LIN {X 0,Y 488.777,Z 238.159,A -85,B 0,C 180,E1 22662.377,E2 22662.377} C_VEL
LIN {X 0,Y 488.746,Z 238.162,A -85,B 0,C 180,E1 22658.896,E2 22658.896} C_VEL
LIN {X 0,Y 488.779,Z 238.165,A -85,B 0,C 180,E1 22655.464,E2 22655.464} C_VEL
LIN {X 0,Y 488.782,Z 238.16,A -85,B 0,C 180,E1 22652.066,E2 22652.066} C_VEL
LIN {X 0,Y 488.749,Z 238.168,A -85,B 0,C 180,E1 22648.693,E2 22648.693} C_VEL
LIN {X 0,Y 488.78,Z 238.161,A -85,B 0,C 180,E1 22645.199,E2 22645.199} C_VEL
LIN {X 0,Y 488.773,Z 238.339,A -85,B 0,C 180,E1 22642.587,E2 22642.587} C_VEL
LIN {X 0,Y 489.136,Z 239.814,A -85,B 0,C 180,E1 22642.324,E2 22642.324} C_VEL
LIN {X 0,Y 490.915,Z 242.687,A -85,B 0,C 180,E1 22641.893,E2 22641.893} C_VEL
LIN {X 0,Y 491.79,Z 244.203,A -85,B 0,C 180,E1 22641.677,E2 22641.677} C_VEL
LIN {X 0,Y 499.359,Z 257.943,A -85,B 0,C 180,E1 22639.854,E2 22639.854} C_VEL
LIN {X 0,Y 508.111,Z 274.612,A -85,B 0,C 180,E1 22637.887,E2 22637.887} C_VEL
LIN {X 0,Y 512.984,Z 283.87,A -85,B 0,C 180,E1 22636.871,E2 22636.871} C_VEL
LIN {X 0,Y 511.655,Z 317.826,A -85,B 0,C 180,E1 22635.138,E2 22635.138} C_VEL
LIN {X 0,Y 513.562,Z 334.327,A -85,B 0,C 180,E1 22634.709,E2 22634.709} C_VEL
LIN {X 0,Y 511.315,Z 543.157,A -85,B 0,C 180,E1 22631.464,E2 22631.464} C_VEL
LIN {X 0,Y 509.844,Z 662.422,A -85,B 0,C 180,E1 22629.623,E2 22629.623} C_VEL
LIN {X 0,Y 508.964,Z 686.115,A -85,B 0,C 180,E1 22629.075,E2 22629.075} C_VEL
LIN {X 0,Y 507.975,Z 706.125,A -85,B 0,C 180,E1 22628.445,E2 22628.445} C_VEL
LIN {X 0,Y 506.503,Z 726.844,A -85,B 0,C 180,E1 22627.586,E2 22627.586} C_VEL
LIN {X 0,Y 504.754,Z 747.351,A -85,B 0,C 180,E1 22626.529,E2 22626.529} C_VEL
LIN {X 0,Y 502.729,Z 769.086,A -85,B 0,C 180,E1 22625.172,E2 22625.172} C_VEL
LIN {X 0,Y 500.805,Z 788.03,A -85,B 0,C 180,E1 22623.78,E2 22623.78} C_VEL
LIN {X 0,Y 498.7,Z 807.609,A -85,B 0,C 180,E1 22622.092,E2 22622.092} C_VEL
LIN {X 0,Y 496.763,Z 825.728,A -85,B 0,C 180,E1 22620.292,E2 22620.292} C_VEL
LIN {X 0,Y 494.892,Z 842.616,A -85,B 0,C 180,E1 22618.344,E2 22618.344} C_VEL
LIN {X 0,Y 493.244,Z 858.757,A -85,B 0,C 180,E1 22616.224,E2 22616.224} C_VEL
LIN {X 0,Y 491.79,Z 873.438,A -85,B 0,C 180,E1 22613.991,E2 22613.991} C_VEL
LIN {X 0,Y 490.472,Z 888.188,A -85,B 0,C 180,E1 22611.4,E2 22611.4} C_VEL
LIN {X 0,Y 489.549,Z 900.169,A -85,B 0,C 180,E1 22608.948,E2 22608.948} C_VEL
LIN {X 0,Y 488.87,Z 910.696,A -85,B 0,C 180,E1 22606.393,E2 22606.393} C_VEL
LIN {X 0,Y 488.409,Z 919.928,A -85,B 0,C 180,E1 22603.736,E2 22603.736} C_VEL
LIN {X 0,Y 488.124,Z 926.96,A -85,B 0,C 180,E1 22601.22,E2 22601.22} C_VEL
LIN {X 0,Y 487.984,Z 932.811,A -85,B 0,C 180,E1 22598.601,E2 22598.601} C_VEL
LIN {X 0,Y 487.929,Z 936.802,A -85,B 0,C 180,E1 22596.116,E2 22596.116} C_VEL
LIN {X 0,Y 487.91,Z 939.633,A -85,B 0,C 180,E1 22593.523,E2 22593.523} C_VEL
LIN {X 0,Y 487.909,Z 940.827,A -85,B 0,C 180,E1 22590.938,E2 22590.938} C_VEL
LIN {X 0,Y 487.9,Z 940.713,A -85,B 0,C 180,E1 22588.472,E2 22588.472} C_VEL
LIN {X 0,Y 487.911,Z 939.068,A -85,B 0,C 180,E1 22585.886,E2 22585.886} C_VEL
LIN {X 0,Y 487.942,Z 936.159,A -85,B 0,C 180,E1 22583.41,E2 22583.41} C_VEL
LIN {X 0,Y 488.024,Z 931.334,A -85,B 0,C 180,E1 22580.684,E2 22580.684} C_VEL
LIN {X 0,Y 488.184,Z 925.576,A -85,B 0,C 180,E1 22578.237,E2 22578.237} C_VEL
LIN {X 0,Y 488.514,Z 917.389,A -85,B 0,C 180,E1 22575.49,E2 22575.49} C_VEL
LIN {X 0,Y 489.013,Z 908.38,A -85,B 0,C 180,E1 22572.998,E2 22572.998} C_VEL
LIN {X 0,Y 489.759,Z 897.294,A -85,B 0,C 180,E1 22570.438,E2 22570.438} C_VEL
LIN {X 0,Y 490.767,Z 884.879,A -85,B 0,C 180,E1 22567.97,E2 22567.97} C_VEL
LIN {X 0,Y 492.003,Z 871.11,A -85,B 0,C 180,E1 22565.634,E2 22565.634} C_VEL
LIN {X 0,Y 493.652,Z 854.64,A -85,B 0,C 180,E1 22563.213,E2 22563.213} C_VEL
LIN {X 0,Y 495.425,Z 838.034,A -85,B 0,C 180,E1 22561.094,E2 22561.094} C_VEL
LIN {X 0,Y 497.321,Z 820.28,A -85,B 0,C 180,E1 22559.146,E2 22559.146} C_VEL
LIN {X 0,Y 499.39,Z 801.44,A -85,B 0,C 180,E1 22557.344,E2 22557.344} C_VEL
LIN {X 0,Y 501.303,Z 783.123,A -85,B 0,C 180,E1 22555.843,E2 22555.843} C_VEL
LIN {X 0,Y 503.334,Z 762.823,A -85,B 0,C 180,E1 22554.405,E2 22554.405} C_VEL
LIN {X 0,Y 505.168,Z 742.786,A -85,B 0,C 180,E1 22553.22,E2 22553.22} C_VEL
LIN {X 0,Y 507.007,Z 720.529,A -85,B 0,C 180,E1 22552.13,E2 22552.13} C_VEL
LIN {X 0,Y 508.179,Z 702.238,A -85,B 0,C 180,E1 22551.421,E2 22551.421} C_VEL
LIN {X 0,Y 509.277,Z 679.493,A -85,B 0,C 180,E1 22550.738,E2 22550.738} C_VEL
LIN {X 0,Y 510.06,Z 656.392,A -85,B 0,C 180,E1 22550.262,E2 22550.262} C_VEL
LIN {X 0,Y 512.708,Z 451.853,A -85,B 0,C 180,E1 22547.063,E2 22547.063} C_VEL
LIN {X 0,Y 514.091,Z 331.525,A -85,B 0,C 180,E1 22545.127,E2 22545.127} C_VEL
LIN {X 0,Y 512.215,Z 314.996,A -85,B 0,C 180,E1 22544.646,E2 22544.646} C_VEL
LIN {X 0,Y 513.652,Z 284.11,A -85,B 0,C 180,E1 22543.022,E2 22543.022} C_VEL
LIN {X 0,Y 502.953,Z 264.154,A -85,B 0,C 180,E1 22540.697,E2 22540.697} C_VEL
LIN {X 0,Y 496.082,Z 251.794,A -85,B 0,C 180,E1 22539.106,E2 22539.106} C_VEL
LIN {X 0,Y 491.249,Z 243.037,A -85,B 0,C 180,E1 22537.928,E2 22537.928} C_VEL
LIN {X 0,Y 489.18,Z 239.919,A -85,B 0,C 180,E1 22537.451,E2 22537.451} C_VEL
LIN {X 0,Y 488.792,Z 238.366,A -85,B 0,C 180,E1 22537.192,E2 22537.192} C_VEL
LIN {X 0,Y 488.759,Z 238.166,A -85,B 0,C 180,E1 22533.632,E2 22533.632} C_VEL
LIN {X 0,Y 488.81,Z 238.16,A -85,B 0,C 180,E1 22530.212,E2 22530.212} C_VEL
LIN {X 0,Y 488.783,Z 238.164,A -85,B 0,C 180,E1 22526.877,E2 22526.877} C_VEL
LIN {X 0,Y 488.768,Z 238.162,A -85,B 0,C 180,E1 22523.382,E2 22523.382} C_VEL
LIN {X 0,Y 488.817,Z 238.157,A -85,B 0,C 180,E1 22519.974,E2 22519.974} C_VEL
LIN {X 0,Y 488.801,Z 238.162,A -85,B 0,C 180,E1 22516.519,E2 22516.519} C_VEL
LIN {X 0,Y 488.777,Z 238.159,A -85,B 0,C 180,E1 22513.125,E2 22513.125} C_VEL
LIN {X 0,Y 488.812,Z 238.151,A -85,B 0,C 180,E1 22509.621,E2 22509.621} C_VEL
LIN {X 0,Y 488.824,Z 238.145,A -85,B 0,C 180,E1 22506.106,E2 22506.106} C_VEL
LIN {X 0,Y 488.79,Z 238.161,A -85,B 0,C 180,E1 22502.58,E2 22502.58} C_VEL
LIN {X 0,Y 488.792,Z 238.158,A -85,B 0,C 180,E1 22498.946,E2 22498.946} C_VEL
LIN {X 0,Y 488.828,Z 238.148,A -85,B 0,C 180,E1 22495.425,E2 22495.425} C_VEL
LIN {X 0,Y 488.826,Z 238.145,A -85,B 0,C 180,E1 22491.887,E2 22491.887} C_VEL
LIN {X 0,Y 488.799,Z 238.159,A -85,B 0,C 180,E1 22488.317,E2 22488.317} C_VEL
LIN {X 0,Y 488.806,Z 238.152,A -85,B 0,C 180,E1 22484.701,E2 22484.701} C_VEL
LIN {X 0,Y 488.829,Z 238.139,A -85,B 0,C 180,E1 22481.146,E2 22481.146} C_VEL
LIN {X 0,Y 488.833,Z 238.155,A -85,B 0,C 180,E1 22477.513,E2 22477.513} C_VEL
LIN {X 0,Y 488.813,Z 238.153,A -85,B 0,C 180,E1 22473.893,E2 22473.893} C_VEL
LIN {X 0,Y 488.812,Z 238.14,A -85,B 0,C 180,E1 22470.331,E2 22470.331} C_VEL
LIN {X 0,Y 488.826,Z 238.15,A -85,B 0,C 180,E1 22466.759,E2 22466.759} C_VEL
LIN {X 0,Y 488.825,Z 238.159,A -85,B 0,C 180,E1 22463.109,E2 22463.109} C_VEL
LIN {X 0,Y 488.82,Z 238.146,A -85,B 0,C 180,E1 22459.545,E2 22459.545} C_VEL
LIN {X 0,Y 488.82,Z 238.144,A -85,B 0,C 180,E1 22455.938,E2 22455.938} C_VEL
LIN {X 0,Y 488.823,Z 238.149,A -85,B 0,C 180,E1 22452.406,E2 22452.406} C_VEL
LIN {X 0,Y 488.818,Z 238.155,A -85,B 0,C 180,E1 22448.75,E2 22448.75} C_VEL
LIN {X 0,Y 488.827,Z 238.159,A -85,B 0,C 180,E1 22445.227,E2 22445.227} C_VEL
LIN {X 0,Y 488.818,Z 238.156,A -85,B 0,C 180,E1 22442.166,E2 22442.166} C_VEL
LIN {X 0,Y 487.85,Z 238.282,A -85,B 0,C 180,E1 22441.263,E2 22441.263} C_VEL
LIN {X 0,Y 481.301,Z 239.095,A -85,B 0,C 180,E1 22438.658,E2 22438.658} C_VEL
LIN {X 0,Y 480.88,Z 239.147,A -85,B 0,C 180,E1 22438.062,E2 22438.062} C_VEL
LIN {X 0,Y 480.87,Z 239.147,A -85,B 0,C 180,E1 22434.397,E2 22434.397} C_VEL
LIN {X 0,Y 480.885,Z 239.102,A -85,B 0,C 180,E1 22430.828,E2 22430.828} C_VEL
LIN {X 0,Y 480.922,Z 239.375,A -85,B 0,C 180,E1 22427.453,E2 22427.453} C_VEL
LIN {X 0,Y 482.307,Z 242.751,A -85,B 0,C 180,E1 22426.935,E2 22426.935} C_VEL
LIN {X 0,Y 483.272,Z 244.312,A -85,B 0,C 180,E1 22426.684,E2 22426.684} C_VEL
LIN {X 0,Y 492.023,Z 261.807,A -85,B 0,C 180,E1 22424.231,E2 22424.231} C_VEL
LIN {X 0,Y 500.621,Z 280.446,A -85,B 0,C 180,E1 22421.866,E2 22421.866} C_VEL
LIN {X 0,Y 500.816,Z 281.709,A -85,B 0,C 180,E1 22421.751,E2 22421.751} C_VEL
LIN {X 0,Y 497.054,Z 336.618,A -85,B 0,C 180,E1 22418.038,E2 22418.038} C_VEL
LIN {X 0,Y 493.768,Z 391.282,A -85,B 0,C 180,E1 22414.414,E2 22414.414} C_VEL
LIN {X 0,Y 492.829,Z 410.278,A -85,B 0,C 180,E1 22413.199,E2 22413.199} C_VEL
LIN {X 0,Y 495.7,Z 434.594,A -85,B 0,C 180,E1 22412.525,E2 22412.525} C_VEL
LIN {X 0,Y 491.917,Z 630.288,A -85,B 0,C 180,E1 22409.324,E2 22409.324} C_VEL
LIN {X 0,Y 491.137,Z 649.987,A -85,B 0,C 180,E1 22408.784,E2 22408.784} C_VEL
LIN {X 0,Y 490.201,Z 668.181,A -85,B 0,C 180,E1 22408.068,E2 22408.068} C_VEL
LIN {X 0,Y 489.059,Z 686.203,A -85,B 0,C 180,E1 22407.13,E2 22407.13} C_VEL
LIN {X 0,Y 487.793,Z 703.294,A -85,B 0,C 180,E1 22406.005,E2 22406.005} C_VEL
LIN {X 0,Y 486.482,Z 719.42,A -85,B 0,C 180,E1 22404.695,E2 22404.695} C_VEL
LIN {X 0,Y 485.186,Z 734.576,A -85,B 0,C 180,E1 22403.196,E2 22403.196} C_VEL
LIN {X 0,Y 483.987,Z 748.249,A -85,B 0,C 180,E1 22401.567,E2 22401.567} C_VEL
LIN {X 0,Y 482.969,Z 760.177,A -85,B 0,C 180,E1 22399.866,E2 22399.866} C_VEL
LIN {X 0,Y 482.049,Z 771.527,A -85,B 0,C 180,E1 22397.909,E2 22397.909} C_VEL
LIN {X 0,Y 481.356,Z 780.906,A -85,B 0,C 180,E1 22395.935,E2 22395.935} C_VEL
LIN {X 0,Y 480.854,Z 788.964,A -85,B 0,C 180,E1 22393.823,E2 22393.823} C_VEL
LIN {X 0,Y 480.512,Z 795.528,A -85,B 0,C 180,E1 22391.593,E2 22391.593} C_VEL
LIN {X 0,Y 480.321,Z 800.233,A -85,B 0,C 180,E1 22389.404,E2 22389.404} C_VEL
LIN {X 0,Y 480.24,Z 803.322,A -85,B 0,C 180,E1 22387.218,E2 22387.218} C_VEL
LIN {X 0,Y 480.207,Z 804.897,A -85,B 0,C 180,E1 22384.92,E2 22384.92} C_VEL
LIN {X 0,Y 480.214,Z 804.804,A -85,B 0,C 180,E1 22382.605,E2 22382.605} C_VEL
LIN {X 0,Y 480.271,Z 803.027,A -85,B 0,C 180,E1 22380.3,E2 22380.3} C_VEL
LIN {X 0,Y 480.393,Z 799.715,A -85,B 0,C 180,E1 22378.087,E2 22378.087} C_VEL
LIN {X 0,Y 480.645,Z 794.619,A -85,B 0,C 180,E1 22375.831,E2 22375.831} C_VEL
LIN {X 0,Y 481.023,Z 788.019,A -85,B 0,C 180,E1 22373.674,E2 22373.674} C_VEL
LIN {X 0,Y 481.584,Z 780.027,A -85,B 0,C 180,E1 22371.629,E2 22371.629} C_VEL
LIN {X 0,Y 482.373,Z 770.427,A -85,B 0,C 180,E1 22369.646,E2 22369.646} C_VEL
LIN {X 0,Y 483.334,Z 759.291,A -85,B 0,C 180,E1 22367.756,E2 22367.756} C_VEL
LIN {X 0,Y 484.484,Z 746.941,A -85,B 0,C 180,E1 22366.019,E2 22366.019} C_VEL
LIN {X 0,Y 485.754,Z 733.257,A -85,B 0,C 180,E1 22364.413,E2 22364.413} C_VEL
LIN {X 0,Y 487.102,Z 718.333,A -85,B 0,C 180,E1 22362.959,E2 22362.959} C_VEL
LIN {X 0,Y 488.479,Z 702.16,A -85,B 0,C 180,E1 22361.662,E2 22361.662} C_VEL
LIN {X 0,Y 489.815,Z 685.013,A -85,B 0,C 180,E1 22360.55,E2 22360.55} C_VEL
LIN {X 0,Y 490.966,Z 667.907,A -85,B 0,C 180,E1 22359.667,E2 22359.667} C_VEL
LIN {X 0,Y 491.994,Z 648.972,A -85,B 0,C 180,E1 22358.927,E2 22358.927} C_VEL
LIN {X 0,Y 492.809,Z 629.599,A -85,B 0,C 180,E1 22358.405,E2 22358.405} C_VEL
LIN {X 0,Y 497.37,Z 433.399,A -85,B 0,C 180,E1 22355.09,E2 22355.09} C_VEL
LIN {X 0,Y 494.063,Z 406.293,A -85,B 0,C 180,E1 22354.235,E2 22354.235} C_VEL
LIN {X 0,Y 497.804,Z 348.948,A -85,B 0,C 180,E1 22350.407,E2 22350.407} C_VEL
LIN {X 0,Y 501.905,Z 294.511,A -85,B 0,C 180,E1 22346.693,E2 22346.693} C_VEL
LIN {X 0,Y 502.643,Z 283.159,A -85,B 0,C 180,E1 22345.888,E2 22345.888} C_VEL
LIN {X 0,Y 494.295,Z 265.385,A -85,B 0,C 180,E1 22343.483,E2 22343.483} C_VEL
LIN {X 0,Y 487.623,Z 252.482,A -85,B 0,C 180,E1 22341.532,E2 22341.532} C_VEL
LIN {X 0,Y 485.062,Z 247.71,A -85,B 0,C 180,E1 22340.765,E2 22340.765} C_VEL
LIN {X 0,Y 482.927,Z 243.642,A -85,B 0,C 180,E1 22340.101,E2 22340.101} C_VEL
LIN {X 0,Y 481.112,Z 240.487,A -85,B 0,C 180,E1 22339.547,E2 22339.547} C_VEL
LIN {X 0,Y 480.861,Z 239.171,A -85,B 0,C 180,E1 22339.226,E2 22339.226} C_VEL
LIN {X 0,Y 480.812,Z 239.157,A -85,B 0,C 180,E1 22335.808,E2 22335.808} C_VEL
LIN {X 0,Y 480.823,Z 239.15,A -85,B 0,C 180,E1 22332.226,E2 22332.226} C_VEL
LIN {X 0,Y 480.874,Z 239.15,A -85,B 0,C 180,E1 22328.73,E2 22328.73} C_VEL
LIN {X 0,Y 480.814,Z 239.15,A -85,B 0,C 180,E1 22325.369,E2 22325.369} C_VEL
LIN {X 0,Y 480.812,Z 239.153,A -85,B 0,C 180,E1 22321.787,E2 22321.787} C_VEL
LIN {X 0,Y 480.871,Z 239.149,A -85,B 0,C 180,E1 22318.451,E2 22318.451} C_VEL
LIN {X 0,Y 480.822,Z 239.155,A -85,B 0,C 180,E1 22314.896,E2 22314.896} C_VEL
LIN {X 0,Y 480.807,Z 239.15,A -85,B 0,C 180,E1 22311.389,E2 22311.389} C_VEL
LIN {X 0,Y 480.846,Z 239.145,A -85,B 0,C 180,E1 22307.876,E2 22307.876} C_VEL
LIN {X 0,Y 480.836,Z 239.146,A -85,B 0,C 180,E1 22304.44,E2 22304.44} C_VEL
LIN {X 0,Y 480.809,Z 239.155,A -85,B 0,C 180,E1 22300.944,E2 22300.944} C_VEL
LIN {X 0,Y 480.828,Z 239.149,A -85,B 0,C 180,E1 22297.405,E2 22297.405} C_VEL
LIN {X 0,Y 480.862,Z 239.145,A -85,B 0,C 180,E1 22293.926,E2 22293.926} C_VEL
LIN {X 0,Y 480.813,Z 239.157,A -85,B 0,C 180,E1 22290.472,E2 22290.472} C_VEL
LIN {X 0,Y 480.814,Z 239.154,A -85,B 0,C 180,E1 22286.844,E2 22286.844} C_VEL
LIN {X 0,Y 480.9,Z 239.379,A -85,B 0,C 180,E1 22283.571,E2 22283.571} C_VEL
LIN {X 0,Y 481.418,Z 241.262,A -85,B 0,C 180,E1 22283.262,E2 22283.262} C_VEL
LIN {X 0,Y 483.785,Z 245.048,A -85,B 0,C 180,E1 22282.657,E2 22282.657} C_VEL
LIN {X 0,Y 489.175,Z 254.643,A -85,B 0,C 180,E1 22281.284,E2 22281.284} C_VEL
LIN {X 0,Y 498.036,Z 270.886,A -85,B 0,C 180,E1 22279.186,E2 22279.186} C_VEL
LIN {X 0,Y 506.549,Z 287.807,A -85,B 0,C 180,E1 22277.268,E2 22277.268} C_VEL
LIN {X 0,Y 505.185,Z 318.867,A -85,B 0,C 180,E1 22275.661,E2 22275.661} C_VEL
LIN {X 0,Y 507.064,Z 335.609,A -85,B 0,C 180,E1 22275.219,E2 22275.219} C_VEL
LIN {X 0,Y 504.613,Z 544.405,A -85,B 0,C 180,E1 22271.943,E2 22271.943} C_VEL
LIN {X 0,Y 503.059,Z 661.873,A -85,B 0,C 180,E1 22270.114,E2 22270.114} C_VEL
LIN {X 0,Y 502.137,Z 685.477,A -85,B 0,C 180,E1 22269.566,E2 22269.566} C_VEL
LIN {X 0,Y 501.063,Z 706.219,A -85,B 0,C 180,E1 22268.91,E2 22268.91} C_VEL
LIN {X 0,Y 499.518,Z 729.104,A -85,B 0,C 180,E1 22267.979,E2 22267.979} C_VEL
LIN {X 0,Y 497.975,Z 749.576,A -85,B 0,C 180,E1 22266.953,E2 22266.953} C_VEL
LIN {X 0,Y 495.997,Z 769.437,A -85,B 0,C 180,E1 22265.694,E2 22265.694} C_VEL
LIN {X 0,Y 493.89,Z 788.838,A -85,B 0,C 180,E1 22264.248,E2 22264.248} C_VEL
LIN {X 0,Y 491.613,Z 808.274,A -85,B 0,C 180,E1 22262.542,E2 22262.542} C_VEL
LIN {X 0,Y 489.506,Z 826.577,A -85,B 0,C 180,E1 22260.691,E2 22260.691} C_VEL
LIN {X 0,Y 487.454,Z 843.629,A -85,B 0,C 180,E1 22258.682,E2 22258.682} C_VEL
LIN {X 0,Y 485.566,Z 860.525,A -85,B 0,C 180,E1 22256.397,E2 22256.397} C_VEL
LIN {X 0,Y 483.993,Z 875.458,A -85,B 0,C 180,E1 22254.062,E2 22254.062} C_VEL
LIN {X 0,Y 482.68,Z 888.821,A -85,B 0,C 180,E1 22251.635,E2 22251.635} C_VEL
LIN {X 0,Y 481.687,Z 900.731,A -85,B 0,C 180,E1 22249.144,E2 22249.144} C_VEL
LIN {X 0,Y 480.948,Z 911.153,A -85,B 0,C 180,E1 22246.546,E2 22246.546} C_VEL
LIN {X 0,Y 480.447,Z 920.285,A -85,B 0,C 180,E1 22243.845,E2 22243.845} C_VEL
LIN {X 0,Y 480.154,Z 926.96,A -85,B 0,C 180,E1 22241.408,E2 22241.408} C_VEL
LIN {X 0,Y 479.991,Z 932.811,A -85,B 0,C 180,E1 22238.745,E2 22238.745} C_VEL
LIN {X 0,Y 479.934,Z 936.801,A -85,B 0,C 180,E1 22236.218,E2 22236.218} C_VEL
LIN {X 0,Y 479.911,Z 939.633,A -85,B 0,C 180,E1 22233.582,E2 22233.582} C_VEL
LIN {X 0,Y 479.909,Z 940.827,A -85,B 0,C 180,E1 22230.954,E2 22230.954} C_VEL
LIN {X 0,Y 479.899,Z 940.713,A -85,B 0,C 180,E1 22228.447,E2 22228.447} C_VEL
LIN {X 0,Y 479.91,Z 939.068,A -85,B 0,C 180,E1 22225.817,E2 22225.817} C_VEL
LIN {X 0,Y 479.944,Z 936.159,A -85,B 0,C 180,E1 22223.299,E2 22223.299} C_VEL
LIN {X 0,Y 480.036,Z 931.334,A -85,B 0,C 180,E1 22220.528,E2 22220.528} C_VEL
LIN {X 0,Y 480.207,Z 925.738,A -85,B 0,C 180,E1 22218.103,E2 22218.103} C_VEL
LIN {X 0,Y 480.573,Z 917.552,A -85,B 0,C 180,E1 22215.295,E2 22215.295} C_VEL
LIN {X 0,Y 481.101,Z 908.845,A -85,B 0,C 180,E1 22212.835,E2 22212.835} C_VEL
LIN {X 0,Y 481.914,Z 897.865,A -85,B 0,C 180,E1 22210.233,E2 22210.233} C_VEL
LIN {X 0,Y 483.014,Z 885.492,A -85,B 0,C 180,E1 22207.715,E2 22207.715} C_VEL
LIN {X 0,Y 484.398,Z 871.306,A -85,B 0,C 180,E1 22205.26,E2 22205.26} C_VEL
LIN {X 0,Y 486.165,Z 855.102,A -85,B 0,C 180,E1 22202.833,E2 22202.833} C_VEL
LIN {X 0,Y 487.975,Z 839.418,A -85,B 0,C 180,E1 22200.794,E2 22200.794} C_VEL
LIN {X 0,Y 490.051,Z 821.594,A -85,B 0,C 180,E1 22198.785,E2 22198.785} C_VEL
LIN {X 0,Y 492.288,Z 802.889,A -85,B 0,C 180,E1 22196.951,E2 22196.951} C_VEL
LIN {X 0,Y 494.501,Z 783.119,A -85,B 0,C 180,E1 22195.306,E2 22195.306} C_VEL
LIN {X 0,Y 496.753,Z 762.204,A -85,B 0,C 180,E1 22193.816,E2 22193.816} C_VEL
LIN {X 0,Y 498.269,Z 745.76,A -85,B 0,C 180,E1 22192.842,E2 22192.842} C_VEL
LIN {X 0,Y 500.018,Z 723.654,A -85,B 0,C 180,E1 22191.764,E2 22191.764} C_VEL
LIN {X 0,Y 501.423,Z 701.01,A -85,B 0,C 180,E1 22190.892,E2 22190.892} C_VEL
LIN {X 0,Y 502.604,Z 677.743,A -85,B 0,C 180,E1 22190.202,E2 22190.202} C_VEL
LIN {X 0,Y 503.42,Z 654.988,A -85,B 0,C 180,E1 22189.736,E2 22189.736} C_VEL
LIN {X 0,Y 506.283,Z 449.649,A -85,B 0,C 180,E1 22186.492,E2 22186.492} C_VEL
LIN {X 0,Y 507.78,Z 332.849,A -85,B 0,C 180,E1 22184.591,E2 22184.591} C_VEL
LIN {X 0,Y 505.905,Z 315.678,A -85,B 0,C 180,E1 22184.082,E2 22184.082} C_VEL
LIN {X 0,Y 507.326,Z 287.949,A -85,B 0,C 180,E1 22182.608,E2 22182.608} C_VEL
LIN {X 0,Y 495.887,Z 266.402,A -85,B 0,C 180,E1 22180.031,E2 22180.031} C_VEL
LIN {X 0,Y 486.035,Z 248.824,A -85,B 0,C 180,E1 22177.661,E2 22177.661} C_VEL
LIN {X 0,Y 483.827,Z 245.145,A -85,B 0,C 180,E1 22177.117,E2 22177.117} C_VEL
LIN {X 0,Y 482.966,Z 243.642,A -85,B 0,C 180,E1 22176.897,E2 22176.897} C_VEL
LIN {X 0,Y 481.046,Z 240.111,A -85,B 0,C 180,E1 22176.381,E2 22176.381} C_VEL
LIN {X 0,Y 480.848,Z 239.202,A -85,B 0,C 180,E1 22176.136,E2 22176.136} C_VEL
LIN {X 0,Y 480.872,Z 239.141,A -85,B 0,C 180,E1 22172.584,E2 22172.584} C_VEL
LIN {X 0,Y 480.83,Z 239.143,A -85,B 0,C 180,E1 22169.117,E2 22169.117} C_VEL
LIN {X 0,Y 480.829,Z 239.141,A -85,B 0,C 180,E1 22165.496,E2 22165.496} C_VEL
LIN {X 0,Y 480.886,Z 239.135,A -85,B 0,C 180,E1 22162.107,E2 22162.107} C_VEL
LIN {X 0,Y 480.85,Z 239.139,A -85,B 0,C 180,E1 22158.677,E2 22158.677} C_VEL
LIN {X 0,Y 480.837,Z 239.144,A -85,B 0,C 180,E1 22155.189,E2 22155.189} C_VEL
LIN {X 0,Y 480.87,Z 239.143,A -85,B 0,C 180,E1 22151.665,E2 22151.665} C_VEL
LIN {X 0,Y 480.887,Z 239.149,A -85,B 0,C 180,E1 22148.128,E2 22148.128} C_VEL
LIN {X 0,Y 480.847,Z 239.142,A -85,B 0,C 180,E1 22144.652,E2 22144.652} C_VEL
LIN {X 0,Y 480.849,Z 239.131,A -85,B 0,C 180,E1 22140.954,E2 22140.954} C_VEL
LIN {X 0,Y 480.889,Z 239.137,A -85,B 0,C 180,E1 22137.498,E2 22137.498} C_VEL
LIN {X 0,Y 480.887,Z 239.147,A -85,B 0,C 180,E1 22133.913,E2 22133.913} C_VEL
LIN {X 0,Y 480.857,Z 239.133,A -85,B 0,C 180,E1 22130.425,E2 22130.425} C_VEL
LIN {X 0,Y 480.867,Z 239.137,A -85,B 0,C 180,E1 22126.779,E2 22126.779} C_VEL
LIN {X 0,Y 480.891,Z 239.145,A -85,B 0,C 180,E1 22123.327,E2 22123.327} C_VEL
LIN {X 0,Y 480.887,Z 239.135,A -85,B 0,C 180,E1 22119.674,E2 22119.674} C_VEL
LIN {X 0,Y 480.868,Z 239.136,A -85,B 0,C 180,E1 22116.081,E2 22116.081} C_VEL
LIN {X 0,Y 480.88,Z 239.144,A -85,B 0,C 180,E1 22112.511,E2 22112.511} C_VEL
LIN {X 0,Y 480.89,Z 239.144,A -85,B 0,C 180,E1 22108.941,E2 22108.941} C_VEL
LIN {X 0,Y 480.887,Z 239.132,A -85,B 0,C 180,E1 22105.272,E2 22105.272} C_VEL
LIN {X 0,Y 480.881,Z 239.141,A -85,B 0,C 180,E1 22101.617,E2 22101.617} C_VEL
LIN {X 0,Y 480.881,Z 239.146,A -85,B 0,C 180,E1 22097.927,E2 22097.927} C_VEL
LIN {X 0,Y 480.888,Z 239.142,A -85,B 0,C 180,E1 22094.316,E2 22094.316} C_VEL
LIN {X 0,Y 480.878,Z 239.137,A -85,B 0,C 180,E1 22090.76,E2 22090.76} C_VEL
LIN {X 0,Y 480.888,Z 239.134,A -85,B 0,C 180,E1 22087.22,E2 22087.22} C_VEL
LIN {X 0,Y 480.885,Z 239.136,A -85,B 0,C 180,E1 22083.579,E2 22083.579} C_VEL
LIN {X 0,Y 480.886,Z 239.134,A -85,B 0,C 180,E1 22079.935,E2 22079.935} C_VEL
LIN {X 0,Y 480.88,Z 239.147,A -85,B 0,C 180,E1 22078.062,E2 22078.062} C_VEL
LIN {X 0,Y 479.908,Z 239.272,A -85,B 0,C 180,E1 22077.144,E2 22077.144} C_VEL
LIN {X 0,Y 473.452,Z 240.076,A -85,B 0,C 180,E1 22074.562,E2 22074.562} C_VEL
LIN {X 0,Y 472.939,Z 240.121,A -85,B 0,C 180,E1 22073.889,E2 22073.889} C_VEL
LIN {X 0,Y 472.924,Z 240.102,A -85,B 0,C 180,E1 22070.289,E2 22070.289} C_VEL
LIN {X 0,Y 472.959,Z 240.33,A -85,B 0,C 180,E1 22068.425,E2 22068.425} C_VEL
LIN {X 0,Y 473.569,Z 242.41,A -85,B 0,C 180,E1 22068.082,E2 22068.082} C_VEL
LIN {X 0,Y 475.472,Z 245.503,A -85,B 0,C 180,E1 22067.565,E2 22067.565} C_VEL
LIN {X 0,Y 483.787,Z 261.827,A -85,B 0,C 180,E1 22065.171,E2 22065.171} C_VEL
LIN {X 0,Y 492.824,Z 281.197,A -85,B 0,C 180,E1 22062.617,E2 22062.617} C_VEL
LIN {X 0,Y 494.338,Z 284.833,A -85,B 0,C 180,E1 22062.177,E2 22062.177} C_VEL
LIN {X 0,Y 490.306,Z 340.338,A -85,B 0,C 180,E1 22058.385,E2 22058.385} C_VEL
LIN {X 0,Y 486.786,Z 395.104,A -85,B 0,C 180,E1 22054.714,E2 22054.714} C_VEL
LIN {X 0,Y 486.045,Z 409.407,A -85,B 0,C 180,E1 22053.794,E2 22053.794} C_VEL
LIN {X 0,Y 489.137,Z 435.737,A -85,B 0,C 180,E1 22053.046,E2 22053.046} C_VEL
LIN {X 0,Y 485.066,Z 630.458,A -85,B 0,C 180,E1 22049.809,E2 22049.809} C_VEL
LIN {X 0,Y 484.231,Z 650.247,A -85,B 0,C 180,E1 22049.262,E2 22049.262} C_VEL
LIN {X 0,Y 483.205,Z 668.858,A -85,B 0,C 180,E1 22048.519,E2 22048.519} C_VEL
LIN {X 0,Y 481.975,Z 686.956,A -85,B 0,C 180,E1 22047.564,E2 22047.564} C_VEL
LIN {X 0,Y 480.615,Z 704.052,A -85,B 0,C 180,E1 22046.423,E2 22046.423} C_VEL
LIN {X 0,Y 479.207,Z 720.197,A -85,B 0,C 180,E1 22045.094,E2 22045.094} C_VEL
LIN {X 0,Y 477.81,Z 735.382,A -85,B 0,C 180,E1 22043.573,E2 22043.573} C_VEL
LIN {X 0,Y 476.511,Z 749.09,A -85,B 0,C 180,E1 22041.92,E2 22041.92} C_VEL
LIN {X 0,Y 475.322,Z 761.808,A -85,B 0,C 180,E1 22040.069,E2 22040.069} C_VEL
LIN {X 0,Y 474.389,Z 772.445,A -85,B 0,C 180,E1 22038.204,E2 22038.204} C_VEL
LIN {X 0,Y 473.616,Z 781.902,A -85,B 0,C 180,E1 22036.191,E2 22036.191} C_VEL
LIN {X 0,Y 473.055,Z 789.968,A -85,B 0,C 180,E1 22034.053,E2 22034.053} C_VEL
LIN {X 0,Y 472.686,Z 796.345,A -85,B 0,C 180,E1 22031.885,E2 22031.885} C_VEL
LIN {X 0,Y 472.448,Z 801.334,A -85,B 0,C 180,E1 22029.563,E2 22029.563} C_VEL
LIN {X 0,Y 472.337,Z 804.595,A -85,B 0,C 180,E1 22027.21,E2 22027.21} C_VEL
LIN {X 0,Y 472.303,Z 806.12,A -85,B 0,C 180,E1 22024.952,E2 22024.952} C_VEL
LIN {X 0,Y 472.311,Z 806.079,A -85,B 0,C 180,E1 22022.655,E2 22022.655} C_VEL
LIN {X 0,Y 472.379,Z 804.375,A -85,B 0,C 180,E1 22020.313,E2 22020.313} C_VEL
LIN {X 0,Y 472.522,Z 801.112,A -85,B 0,C 180,E1 22018.049,E2 22018.049} C_VEL
LIN {X 0,Y 472.804,Z 796.132,A -85,B 0,C 180,E1 22015.772,E2 22015.772} C_VEL
LIN {X 0,Y 473.226,Z 789.632,A -85,B 0,C 180,E1 22013.581,E2 22013.581} C_VEL
LIN {X 0,Y 473.889,Z 781.092,A -85,B 0,C 180,E1 22011.354,E2 22011.354} C_VEL
LIN {X 0,Y 474.781,Z 771.251,A -85,B 0,C 180,E1 22009.299,E2 22009.299} C_VEL
LIN {X 0,Y 475.872,Z 759.784,A -85,B 0,C 180,E1 22007.339,E2 22007.339} C_VEL
LIN {X 0,Y 477.133,Z 747.372,A -85,B 0,C 180,E1 22005.582,E2 22005.582} C_VEL
LIN {X 0,Y 478.548,Z 733.249,A -85,B 0,C 180,E1 22003.92,E2 22003.92} C_VEL
LIN {X 0,Y 480.025,Z 718.096,A -85,B 0,C 180,E1 22002.443,E2 22002.443} C_VEL
LIN {X 0,Y 481.469,Z 702.264,A -85,B 0,C 180,E1 22001.17,E2 22001.17} C_VEL
LIN {X 0,Y 482.899,Z 685.05,A -85,B 0,C 180,E1 22000.047,E2 22000.047} C_VEL
LIN {X 0,Y 484.146,Z 667.79,A -85,B 0,C 180,E1 21999.154,E2 21999.154} C_VEL
LIN {X 0,Y 485.223,Z 649.251,A -85,B 0,C 180,E1 21998.424,E2 21998.424} C_VEL
LIN {X 0,Y 486.092,Z 629.922,A -85,B 0,C 180,E1 21997.896,E2 21997.896} C_VEL
LIN {X 0,Y 491.068,Z 435.005,A -85,B 0,C 180,E1 21994.548,E2 21994.548} C_VEL
LIN {X 0,Y 487.47,Z 405.253,A -85,B 0,C 180,E1 21993.596,E2 21993.596} C_VEL
LIN {X 0,Y 491.519,Z 347.723,A -85,B 0,C 180,E1 21989.706,E2 21989.706} C_VEL
LIN {X 0,Y 496.008,Z 292.314,A -85,B 0,C 180,E1 21985.875,E2 21985.875} C_VEL
LIN {X 0,Y 496.429,Z 287.412,A -85,B 0,C 180,E1 21985.531,E2 21985.531} C_VEL
LIN {X 0,Y 488.348,Z 270.131,A -85,B 0,C 180,E1 21983.147,E2 21983.147} C_VEL
LIN {X 0,Y 482.137,Z 257.93,A -85,B 0,C 180,E1 21981.279,E2 21981.279} C_VEL
LIN {X 0,Y 477.474,Z 249.219,A -85,B 0,C 180,E1 21979.83,E2 21979.83} C_VEL
LIN {X 0,Y 475.053,Z 244.639,A -85,B 0,C 180,E1 21979.04,E2 21979.04} C_VEL
LIN {X 0,Y 473.234,Z 241.662,A -85,B 0,C 180,E1 21978.476,E2 21978.476} C_VEL
LIN {X 0,Y 472.881,Z 240.189,A -85,B 0,C 180,E1 21978.128,E2 21978.128} C_VEL
LIN {X 0,Y 472.92,Z 240.134,A -85,B 0,C 180,E1 21974.696,E2 21974.696} C_VEL
LIN {X 0,Y 472.9,Z 240.144,A -85,B 0,C 180,E1 21971.185,E2 21971.185} C_VEL
LIN {X 0,Y 472.87,Z 240.137,A -85,B 0,C 180,E1 21967.655,E2 21967.655} C_VEL
LIN {X 0,Y 472.89,Z 240.144,A -85,B 0,C 180,E1 21964.122,E2 21964.122} C_VEL
LIN {X 0,Y 472.937,Z 240.134,A -85,B 0,C 180,E1 21960.523,E2 21960.523} C_VEL
LIN {X 0,Y 472.883,Z 240.137,A -85,B 0,C 180,E1 21956.97,E2 21956.97} C_VEL
LIN {X 0,Y 472.87,Z 240.138,A -85,B 0,C 180,E1 21953.443,E2 21953.443} C_VEL
LIN {X 0,Y 472.915,Z 240.137,A -85,B 0,C 180,E1 21950.016,E2 21950.016} C_VEL
LIN {X 0,Y 472.905,Z 240.142,A -85,B 0,C 180,E1 21946.427,E2 21946.427} C_VEL
LIN {X 0,Y 472.87,Z 240.143,A -85,B 0,C 180,E1 21942.908,E2 21942.908} C_VEL
LIN {X 0,Y 472.88,Z 240.136,A -85,B 0,C 180,E1 21939.322,E2 21939.322} C_VEL
LIN {X 0,Y 472.929,Z 240.135,A -85,B 0,C 180,E1 21935.918,E2 21935.918} C_VEL
LIN {X 0,Y 472.882,Z 240.142,A -85,B 0,C 180,E1 21932.362,E2 21932.362} C_VEL
LIN {X 0,Y 472.873,Z 240.144,A -85,B 0,C 180,E1 21928.799,E2 21928.799} C_VEL
LIN {X 0,Y 472.913,Z 240.136,A -85,B 0,C 180,E1 21925.327,E2 21925.327} C_VEL
LIN {X 0,Y 472.894,Z 240.287,A -85,B 0,C 180,E1 21924.697,E2 21924.697} C_VEL
LIN {X 0,Y 473.134,Z 241.408,A -85,B 0,C 180,E1 21924.447,E2 21924.447} C_VEL
LIN {X 0,Y 475.106,Z 244.733,A -85,B 0,C 180,E1 21923.895,E2 21923.895} C_VEL
LIN {X 0,Y 475.962,Z 246.044,A -85,B 0,C 180,E1 21923.672,E2 21923.672} C_VEL
LIN {X 0,Y 478.251,Z 249.957,A -85,B 0,C 180,E1 21923.054,E2 21923.054} C_VEL
LIN {X 0,Y 486.613,Z 265.068,A -85,B 0,C 180,E1 21920.891,E2 21920.891} C_VEL
LIN {X 0,Y 495.628,Z 282.43,A -85,B 0,C 180,E1 21918.725,E2 21918.725} C_VEL
LIN {X 0,Y 500.147,Z 291.325,A -85,B 0,C 180,E1 21917.701,E2 21917.701} C_VEL
LIN {X 0,Y 498.795,Z 319.968,A -85,B 0,C 180,E1 21916.201,E2 21916.201} C_VEL
LIN {X 0,Y 500.621,Z 336.934,A -85,B 0,C 180,E1 21915.744,E2 21915.744} C_VEL
LIN {X 0,Y 497.95,Z 545.494,A -85,B 0,C 180,E1 21912.439,E2 21912.439} C_VEL
LIN {X 0,Y 496.311,Z 661.746,A -85,B 0,C 180,E1 21910.612,E2 21910.612} C_VEL
LIN {X 0,Y 495.334,Z 685.117,A -85,B 0,C 180,E1 21910.064,E2 21910.064} C_VEL
LIN {X 0,Y 494.177,Z 706.236,A -85,B 0,C 180,E1 21909.389,E2 21909.389} C_VEL
LIN {X 0,Y 492.587,Z 728.496,A -85,B 0,C 180,E1 21908.47,E2 21908.47} C_VEL
LIN {X 0,Y 490.85,Z 750.217,A -85,B 0,C 180,E1 21907.373,E2 21907.373} C_VEL
LIN {X 0,Y 488.918,Z 771.146,A -85,B 0,C 180,E1 21906.082,E2 21906.082} C_VEL
LIN {X 0,Y 487.368,Z 786.381,A -85,B 0,C 180,E1 21904.986,E2 21904.986} C_VEL
LIN {X 0,Y 484.824,Z 806.913,A -85,B 0,C 180,E1 21903.199,E2 21903.199} C_VEL
LIN {X 0,Y 482.596,Z 824.72,A -85,B 0,C 180,E1 21901.395,E2 21901.395} C_VEL
LIN {X 0,Y 480.36,Z 842.108,A -85,B 0,C 180,E1 21899.351,E2 21899.351} C_VEL
LIN {X 0,Y 478.452,Z 857.894,A -85,B 0,C 180,E1 21897.235,E2 21897.235} C_VEL
LIN {X 0,Y 476.685,Z 872.664,A -85,B 0,C 180,E1 21894.934,E2 21894.934} C_VEL
LIN {X 0,Y 475.17,Z 886.911,A -85,B 0,C 180,E1 21892.385,E2 21892.385} C_VEL
LIN {X 0,Y 474.071,Z 898.445,A -85,B 0,C 180,E1 21889.977,E2 21889.977} C_VEL
LIN {X 0,Y 473.157,Z 909.776,A -85,B 0,C 180,E1 21887.207,E2 21887.207} C_VEL
LIN {X 0,Y 472.604,Z 918.37,A -85,B 0,C 180,E1 21884.706,E2 21884.706} C_VEL
LIN {X 0,Y 472.226,Z 926.05,A -85,B 0,C 180,E1 21881.974,E2 21881.974} C_VEL
LIN {X 0,Y 472.039,Z 931.848,A -85,B 0,C 180,E1 21879.385,E2 21879.385} C_VEL
LIN {X 0,Y 471.944,Z 936.482,A -85,B 0,C 180,E1 21876.568,E2 21876.568} C_VEL
LIN {X 0,Y 471.912,Z 939.296,A -85,B 0,C 180,E1 21874.008,E2 21874.008} C_VEL
LIN {X 0,Y 471.912,Z 940.782,A -85,B 0,C 180,E1 21871.213,E2 21871.213} C_VEL
LIN {X 0,Y 471.912,Z 940.781,A -85,B 0,C 180,E1 21868.785,E2 21868.785} C_VEL
LIN {X 0,Y 471.913,Z 939.294,A -85,B 0,C 180,E1 21865.989,E2 21865.989} C_VEL
LIN {X 0,Y 471.944,Z 936.478,A -85,B 0,C 180,E1 21863.43,E2 21863.43} C_VEL
LIN {X 0,Y 472.039,Z 931.842,A -85,B 0,C 180,E1 21860.612,E2 21860.612} C_VEL
LIN {X 0,Y 472.228,Z 926.022,A -85,B 0,C 180,E1 21858.015,E2 21858.015} C_VEL
LIN {X 0,Y 472.625,Z 917.956,A -85,B 0,C 180,E1 21855.167,E2 21855.167} C_VEL
LIN {X 0,Y 473.193,Z 909.31,A -85,B 0,C 180,E1 21852.665,E2 21852.665} C_VEL
LIN {X 0,Y 474.122,Z 897.864,A -85,B 0,C 180,E1 21849.894,E2 21849.894} C_VEL
LIN {X 0,Y 475.317,Z 885.613,A -85,B 0,C 180,E1 21847.358,E2 21847.358} C_VEL
LIN {X 0,Y 476.772,Z 871.877,A -85,B 0,C 180,E1 21844.935,E2 21844.935} C_VEL
LIN {X 0,Y 478.564,Z 856.824,A -85,B 0,C 180,E1 21842.616,E2 21842.616} C_VEL
LIN {X 0,Y 480.501,Z 841.074,A -85,B 0,C 180,E1 21840.519,E2 21840.519} C_VEL
LIN {X 0,Y 482.905,Z 822.015,A -85,B 0,C 180,E1 21838.318,E2 21838.318} C_VEL
LIN {X 0,Y 485.285,Z 803.563,A -85,B 0,C 180,E1 21836.483,E2 21836.483} C_VEL
LIN {X 0,Y 487.547,Z 784.684,A -85,B 0,C 180,E1 21834.882,E2 21834.882} C_VEL
LIN {X 0,Y 489.376,Z 766.616,A -85,B 0,C 180,E1 21833.61,E2 21833.61} C_VEL
LIN {X 0,Y 491.346,Z 745.051,A -85,B 0,C 180,E1 21832.334,E2 21832.334} C_VEL
LIN {X 0,Y 493.122,Z 723.818,A -85,B 0,C 180,E1 21831.286,E2 21831.286} C_VEL
LIN {X 0,Y 494.636,Z 701.135,A -85,B 0,C 180,E1 21830.397,E2 21830.397} C_VEL
LIN {X 0,Y 495.903,Z 678.074,A -85,B 0,C 180,E1 21829.7,E2 21829.7} C_VEL
LIN {X 0,Y 496.776,Z 655.142,A -85,B 0,C 180,E1 21829.224,E2 21829.224} C_VEL
LIN {X 0,Y 499.879,Z 449.56,A -85,B 0,C 180,E1 21825.941,E2 21825.941} C_VEL
LIN {X 0,Y 501.515,Z 334.17,A -85,B 0,C 180,E1 21824.041,E2 21824.041} C_VEL
LIN {X 0,Y 499.642,Z 316.366,A -85,B 0,C 180,E1 21823.503,E2 21823.503} C_VEL
LIN {X 0,Y 501.048,Z 291.884,A -85,B 0,C 180,E1 21822.19,E2 21822.19} C_VEL
LIN {X 0,Y 490.636,Z 272.058,A -85,B 0,C 180,E1 21819.784,E2 21819.784} C_VEL
LIN {X 0,Y 480.85,Z 254.542,A -85,B 0,C 180,E1 21817.385,E2 21817.385} C_VEL
LIN {X 0,Y 475.903,Z 245.94,A -85,B 0,C 180,E1 21816.109,E2 21816.109} C_VEL
LIN {X 0,Y 473.461,Z 242.298,A -85,B 0,C 180,E1 21815.503,E2 21815.503} C_VEL
LIN {X 0,Y 472.932,Z 240.454,A -85,B 0,C 180,E1 21815.213,E2 21815.213} C_VEL
LIN {X 0,Y 472.9,Z 240.134,A -85,B 0,C 180,E1 21814.022,E2 21814.022} C_VEL
LIN {X 0,Y 472.948,Z 240.138,A -85,B 0,C 180,E1 21810.394,E2 21810.394} C_VEL
LIN {X 0,Y 472.907,Z 240.139,A -85,B 0,C 180,E1 21806.844,E2 21806.844} C_VEL
LIN {X 0,Y 472.89,Z 240.141,A -85,B 0,C 180,E1 21803.29,E2 21803.29} C_VEL
LIN {X 0,Y 472.92,Z 240.135,A -85,B 0,C 180,E1 21799.772,E2 21799.772} C_VEL
LIN {X 0,Y 472.949,Z 240.135,A -85,B 0,C 180,E1 21796.204,E2 21796.204} C_VEL
LIN {X 0,Y 472.907,Z 240.138,A -85,B 0,C 180,E1 21792.703,E2 21792.703} C_VEL
LIN {X 0,Y 472.905,Z 240.134,A -85,B 0,C 180,E1 21789.111,E2 21789.111} C_VEL
LIN {X 0,Y 472.94,Z 240.121,A -85,B 0,C 180,E1 21785.581,E2 21785.581} C_VEL
LIN {X 0,Y 472.948,Z 240.121,A -85,B 0,C 180,E1 21781.939,E2 21781.939} C_VEL
LIN {X 0,Y 472.918,Z 240.139,A -85,B 0,C 180,E1 21778.425,E2 21778.425} C_VEL
LIN {X 0,Y 472.915,Z 240.131,A -85,B 0,C 180,E1 21774.758,E2 21774.758} C_VEL
LIN {X 0,Y 472.946,Z 240.116,A -85,B 0,C 180,E1 21771.245,E2 21771.245} C_VEL
LIN {X 0,Y 472.952,Z 240.129,A -85,B 0,C 180,E1 21767.612,E2 21767.612} C_VEL
LIN {X 0,Y 472.931,Z 240.133,A -85,B 0,C 180,E1 21764.048,E2 21764.048} C_VEL
LIN {X 0,Y 472.925,Z 240.117,A -85,B 0,C 180,E1 21760.358,E2 21760.358} C_VEL
LIN {X 0,Y 472.945,Z 240.126,A -85,B 0,C 180,E1 21756.714,E2 21756.714} C_VEL
LIN {X 0,Y 472.951,Z 240.135,A -85,B 0,C 180,E1 21753.102,E2 21753.102} C_VEL
LIN {X 0,Y 472.955,Z 240.12,A -85,B 0,C 180,E1 21749.512,E2 21749.512} C_VEL
LIN {X 0,Y 472.934,Z 240.125,A -85,B 0,C 180,E1 21745.928,E2 21745.928} C_VEL
LIN {X 0,Y 472.945,Z 240.133,A -85,B 0,C 180,E1 21742.25,E2 21742.25} C_VEL
LIN {X 0,Y 472.948,Z 240.133,A -85,B 0,C 180,E1 21738.57,E2 21738.57} C_VEL
LIN {X 0,Y 472.944,Z 240.126,A -85,B 0,C 180,E1 21734.91,E2 21734.91} C_VEL
LIN {X 0,Y 472.955,Z 240.12,A -85,B 0,C 180,E1 21731.184,E2 21731.184} C_VEL
LIN {X 0,Y 472.943,Z 240.123,A -85,B 0,C 180,E1 21727.509,E2 21727.509} C_VEL
LIN {X 0,Y 472.951,Z 240.125,A -85,B 0,C 180,E1 21723.817,E2 21723.817} C_VEL
LIN {X 0,Y 472.937,Z 240.125,A -85,B 0,C 180,E1 21720.155,E2 21720.155} C_VEL
LIN {X 0,Y 472.932,Z 240.125,A -85,B 0,C 180,E1 21716.494,E2 21716.494} C_VEL
LIN {X 0,Y 472.939,Z 240.121,A -85,B 0,C 180,E1 21713.889,E2 21713.889} C_VEL
LIN {X 0,Y 471.971,Z 240.226,A -85,B 0,C 180,E1 21712.955,E2 21712.955} C_VEL
LIN {X 0,Y 465.423,Z 241.036,A -85,B 0,C 180,E1 21710.262,E2 21710.262} C_VEL
LIN {X 0,Y 465.007,Z 241.117,A -85,B 0,C 180,E1 21709.645,E2 21709.645} C_VEL
LIN {X 0,Y 465.11,Z 241.711,A -85,B 0,C 180,E1 21709.315,E2 21709.315} C_VEL
LIN {X 0,Y 466.784,Z 245.229,A -85,B 0,C 180,E1 21708.743,E2 21708.743} C_VEL
LIN {X 0,Y 472.22,Z 255.491,A -85,B 0,C 180,E1 21707.117,E2 21707.117} C_VEL
LIN {X 0,Y 480.487,Z 272.136,A -85,B 0,C 180,E1 21704.708,E2 21704.708} C_VEL
LIN {X 0,Y 487.859,Z 288.348,A -85,B 0,C 180,E1 21702.587,E2 21702.587} C_VEL
LIN {X 0,Y 483.628,Z 343.169,A -85,B 0,C 180,E1 21698.801,E2 21698.801} C_VEL
LIN {X 0,Y 479.874,Z 398.05,A -85,B 0,C 180,E1 21695.082,E2 21695.082} C_VEL
LIN {X 0,Y 479.337,Z 408.729,A -85,B 0,C 180,E1 21694.399,E2 21694.399} C_VEL
LIN {X 0,Y 482.618,Z 436.875,A -85,B 0,C 180,E1 21693.581,E2 21693.581} C_VEL
LIN {X 0,Y 478.243,Z 630.835,A -85,B 0,C 180,E1 21690.304,E2 21690.304} C_VEL
LIN {X 0,Y 477.346,Z 650.716,A -85,B 0,C 180,E1 21689.746,E2 21689.746} C_VEL
LIN {X 0,Y 476.233,Z 669.638,A -85,B 0,C 180,E1 21688.979,E2 21688.979} C_VEL
LIN {X 0,Y 474.895,Z 687.984,A -85,B 0,C 180,E1 21687.993,E2 21687.993} C_VEL
LIN {X 0,Y 473.465,Z 704.809,A -85,B 0,C 180,E1 21686.854,E2 21686.854} C_VEL
LIN {X 0,Y 471.958,Z 720.972,A -85,B 0,C 180,E1 21685.506,E2 21685.506} C_VEL
LIN {X 0,Y 470.498,Z 735.809,A -85,B 0,C 180,E1 21684.006,E2 21684.006} C_VEL
LIN {X 0,Y 469.054,Z 749.929,A -85,B 0,C 180,E1 21682.284,E2 21682.284} C_VEL
LIN {X 0,Y 467.763,Z 762.688,A -85,B 0,C 180,E1 21680.404,E2 21680.404} C_VEL
LIN {X 0,Y 466.678,Z 773.992,A -85,B 0,C 180,E1 21678.383,E2 21678.383} C_VEL
LIN {X 0,Y 465.846,Z 783.337,A -85,B 0,C 180,E1 21676.345,E2 21676.345} C_VEL
LIN {X 0,Y 465.23,Z 791.378,A -85,B 0,C 180,E1 21674.162,E2 21674.162} C_VEL
LIN {X 0,Y 464.822,Z 797.732,A -85,B 0,C 180,E1 21671.943,E2 21671.943} C_VEL
LIN {X 0,Y 464.56,Z 802.643,A -85,B 0,C 180,E1 21669.596,E2 21669.596} C_VEL
LIN {X 0,Y 464.445,Z 805.745,A -85,B 0,C 180,E1 21667.336,E2 21667.336} C_VEL
LIN {X 0,Y 464.399,Z 807.336,A -85,B 0,C 180,E1 21665.013,E2 21665.013} C_VEL
LIN {X 0,Y 464.409,Z 807.354,A -85,B 0,C 180,E1 21662.706,E2 21662.706} C_VEL
LIN {X 0,Y 464.486,Z 805.721,A -85,B 0,C 180,E1 21660.325,E2 21660.325} C_VEL
LIN {X 0,Y 464.654,Z 802.439,A -85,B 0,C 180,E1 21657.974,E2 21657.974} C_VEL
LIN {X 0,Y 464.97,Z 797.516,A -85,B 0,C 180,E1 21655.662,E2 21655.662} C_VEL
LIN {X 0,Y 465.464,Z 790.724,A -85,B 0,C 180,E1 21653.335,E2 21653.335} C_VEL
LIN {X 0,Y 466.186,Z 782.403,A -85,B 0,C 180,E1 21651.126,E2 21651.126} C_VEL
LIN {X 0,Y 467.145,Z 772.778,A -85,B 0,C 180,E1 21649.072,E2 21649.072} C_VEL
LIN {X 0,Y 468.329,Z 761.366,A -85,B 0,C 180,E1 21647.077,E2 21647.077} C_VEL
LIN {X 0,Y 469.665,Z 749.251,A -85,B 0,C 180,E1 21645.319,E2 21645.319} C_VEL
LIN {X 0,Y 471.209,Z 734.994,A -85,B 0,C 180,E1 21643.599,E2 21643.599} C_VEL
LIN {X 0,Y 472.811,Z 719.764,A -85,B 0,C 180,E1 21642.078,E2 21642.078} C_VEL
LIN {X 0,Y 474.41,Z 703.503,A -85,B 0,C 180,E1 21640.743,E2 21640.743} C_VEL
LIN {X 0,Y 475.936,Z 686.416,A -85,B 0,C 180,E1 21639.606,E2 21639.606} C_VEL
LIN {X 0,Y 477.312,Z 668.595,A -85,B 0,C 180,E1 21638.667,E2 21638.667} C_VEL
LIN {X 0,Y 478.476,Z 649.87,A -85,B 0,C 180,E1 21637.918,E2 21637.918} C_VEL
LIN {X 0,Y 479.41,Z 630.455,A -85,B 0,C 180,E1 21637.378,E2 21637.378} C_VEL
LIN {X 0,Y 484.359,Z 450.771,A -85,B 0,C 180,E1 21634.234,E2 21634.234} C_VEL
LIN {X 0,Y 484.618,Z 434.99,A -85,B 0,C 180,E1 21633.941,E2 21633.941} C_VEL
LIN {X 0,Y 480.941,Z 404.111,A -85,B 0,C 180,E1 21632.931,E2 21632.931} C_VEL
LIN {X 0,Y 485.246,Z 347.221,A -85,B 0,C 180,E1 21629.035,E2 21629.035} C_VEL
LIN {X 0,Y 490.108,Z 291.144,A -85,B 0,C 180,E1 21625.108,E2 21625.108} C_VEL
LIN {X 0,Y 482.078,Z 274.102,A -85,B 0,C 180,E1 21622.691,E2 21622.691} C_VEL
LIN {X 0,Y 476.31,Z 262.742,A -85,B 0,C 180,E1 21620.907,E2 21620.907} C_VEL
LIN {X 0,Y 471.698,Z 254.158,A -85,B 0,C 180,E1 21619.438,E2 21619.438} C_VEL
LIN {X 0,Y 469.651,Z 250.244,A -85,B 0,C 180,E1 21618.751,E2 21618.751} C_VEL
LIN {X 0,Y 467.265,Z 245.851,A -85,B 0,C 180,E1 21617.946,E2 21617.946} C_VEL
LIN {X 0,Y 465.461,Z 243.088,A -85,B 0,C 180,E1 21617.372,E2 21617.372} C_VEL
LIN {X 0,Y 465.032,Z 241.432,A -85,B 0,C 180,E1 21617.066,E2 21617.066} C_VEL
LIN {X 0,Y 464.949,Z 241.134,A -85,B 0,C 180,E1 21615.465,E2 21615.465} C_VEL
LIN {X 0,Y 464.934,Z 241.13,A -85,B 0,C 180,E1 21611.913,E2 21611.913} C_VEL
LIN {X 0,Y 464.968,Z 241.126,A -85,B 0,C 180,E1 21608.408,E2 21608.408} C_VEL
LIN {X 0,Y 464.966,Z 241.123,A -85,B 0,C 180,E1 21604.934,E2 21604.934} C_VEL
LIN {X 0,Y 464.934,Z 241.132,A -85,B 0,C 180,E1 21601.355,E2 21601.355} C_VEL
LIN {X 0,Y 464.935,Z 241.13,A -85,B 0,C 180,E1 21597.658,E2 21597.658} C_VEL
LIN {X 0,Y 464.984,Z 241.12,A -85,B 0,C 180,E1 21594.199,E2 21594.199} C_VEL
LIN {X 0,Y 464.95,Z 241.123,A -85,B 0,C 180,E1 21590.718,E2 21590.718} C_VEL
LIN {X 0,Y 464.931,Z 241.13,A -85,B 0,C 180,E1 21587.202,E2 21587.202} C_VEL
LIN {X 0,Y 464.969,Z 241.132,A -85,B 0,C 180,E1 21583.766,E2 21583.766} C_VEL
LIN {X 0,Y 464.98,Z 241.125,A -85,B 0,C 180,E1 21580.138,E2 21580.138} C_VEL
LIN {X 0,Y 464.935,Z 241.125,A -85,B 0,C 180,E1 21576.671,E2 21576.671} C_VEL
LIN {X 0,Y 464.935,Z 241.135,A -85,B 0,C 180,E1 21572.91,E2 21572.91} C_VEL
LIN {X 0,Y 464.967,Z 241.124,A -85,B 0,C 180,E1 21569.36,E2 21569.36} C_VEL
LIN {X 0,Y 464.988,Z 241.264,A -85,B 0,C 180,E1 21565.859,E2 21565.859} C_VEL
LIN {X 0,Y 465.269,Z 242.446,A -85,B 0,C 180,E1 21565.585,E2 21565.585} C_VEL
LIN {X 0,Y 467.193,Z 245.761,A -85,B 0,C 180,E1 21565.001,E2 21565.001} C_VEL
LIN {X 0,Y 468.021,Z 246.966,A -85,B 0,C 180,E1 21564.773,E2 21564.773} C_VEL
LIN {X 0,Y 469.971,Z 250.524,A -85,B 0,C 180,E1 21564.193,E2 21564.193} C_VEL
LIN {X 0,Y 471.218,Z 252.585,A -85,B 0,C 180,E1 21563.852,E2 21563.852} C_VEL
LIN {X 0,Y 478.369,Z 265.091,A -85,B 0,C 180,E1 21561.932,E2 21561.932} C_VEL
LIN {X 0,Y 487.598,Z 282.602,A -85,B 0,C 180,E1 21559.61,E2 21559.61} C_VEL
LIN {X 0,Y 493.782,Z 295.482,A -85,B 0,C 180,E1 21558.109,E2 21558.109} C_VEL
LIN {X 0,Y 492.445,Z 321.048,A -85,B 0,C 180,E1 21556.755,E2 21556.755} C_VEL
LIN {X 0,Y 494.243,Z 338.132,A -85,B 0,C 180,E1 21556.288,E2 21556.288} C_VEL
LIN {X 0,Y 491.336,Z 545.881,A -85,B 0,C 180,E1 21552.958,E2 21552.958} C_VEL
LIN {X 0,Y 489.601,Z 661.744,A -85,B 0,C 180,E1 21551.121,E2 21551.121} C_VEL
LIN {X 0,Y 488.57,Z 684.76,A -85,B 0,C 180,E1 21550.575,E2 21550.575} C_VEL
LIN {X 0,Y 487.334,Z 706.129,A -85,B 0,C 180,E1 21549.885,E2 21549.885} C_VEL
LIN {X 0,Y 485.651,Z 728.328,A -85,B 0,C 180,E1 21548.955,E2 21548.955} C_VEL
LIN {X 0,Y 483.825,Z 749.729,A -85,B 0,C 180,E1 21547.861,E2 21547.861} C_VEL
LIN {X 0,Y 481.771,Z 770.613,A -85,B 0,C 180,E1 21546.556,E2 21546.556} C_VEL
LIN {X 0,Y 479.609,Z 791.454,A -85,B 0,C 180,E1 21545.033,E2 21545.033} C_VEL
LIN {X 0,Y 477.617,Z 808.811,A -85,B 0,C 180,E1 21543.548,E2 21543.548} C_VEL
LIN {X 0,Y 475.592,Z 824.05,A -85,B 0,C 180,E1 21541.989,E2 21541.989} C_VEL
LIN {X 0,Y 473.199,Z 841.601,A -85,B 0,C 180,E1 21539.91,E2 21539.91} C_VEL
LIN {X 0,Y 471.041,Z 857.893,A -85,B 0,C 180,E1 21537.699,E2 21537.699} C_VEL
LIN {X 0,Y 469.134,Z 872.704,A -85,B 0,C 180,E1 21535.356,E2 21535.356} C_VEL
LIN {X 0,Y 467.494,Z 886.912,A -85,B 0,C 180,E1 21532.773,E2 21532.773} C_VEL
LIN {X 0,Y 466.283,Z 898.443,A -85,B 0,C 180,E1 21530.326,E2 21530.326} C_VEL
LIN {X 0,Y 465.287,Z 909.774,A -85,B 0,C 180,E1 21527.507,E2 21527.507} C_VEL
LIN {X 0,Y 464.677,Z 918.39,A -85,B 0,C 180,E1 21524.956,E2 21524.956} C_VEL
LIN {X 0,Y 464.25,Z 926.249,A -85,B 0,C 180,E1 21522.1,E2 21522.1} C_VEL
LIN {X 0,Y 464.046,Z 932.102,A -85,B 0,C 180,E1 21519.423,E2 21519.423} C_VEL
LIN {X 0,Y 463.946,Z 936.482,A -85,B 0,C 180,E1 21516.682,E2 21516.682} C_VEL
LIN {X 0,Y 463.912,Z 939.297,A -85,B 0,C 180,E1 21514.077,E2 21514.077} C_VEL
LIN {X 0,Y 463.911,Z 940.781,A -85,B 0,C 180,E1 21511.234,E2 21511.234} C_VEL
LIN {X 0,Y 463.911,Z 940.781,A -85,B 0,C 180,E1 21508.764,E2 21508.764} C_VEL
LIN {X 0,Y 463.913,Z 939.294,A -85,B 0,C 180,E1 21505.92,E2 21505.92} C_VEL
LIN {X 0,Y 463.947,Z 936.478,A -85,B 0,C 180,E1 21503.316,E2 21503.316} C_VEL
LIN {X 0,Y 464.049,Z 931.842,A -85,B 0,C 180,E1 21500.449,E2 21500.449} C_VEL
LIN {X 0,Y 464.257,Z 926.042,A -85,B 0,C 180,E1 21497.814,E2 21497.814} C_VEL
LIN {X 0,Y 464.703,Z 917.955,A -85,B 0,C 180,E1 21494.908,E2 21494.908} C_VEL
LIN {X 0,Y 465.326,Z 909.31,A -85,B 0,C 180,E1 21492.363,E2 21492.363} C_VEL
LIN {X 0,Y 466.333,Z 897.862,A -85,B 0,C 180,E1 21489.543,E2 21489.543} C_VEL
LIN {X 0,Y 467.645,Z 885.615,A -85,B 0,C 180,E1 21486.966,E2 21486.966} C_VEL
LIN {X 0,Y 469.238,Z 871.875,A -85,B 0,C 180,E1 21484.504,E2 21484.504} C_VEL
LIN {X 0,Y 471.186,Z 856.61,A -85,B 0,C 180,E1 21482.119,E2 21482.119} C_VEL
LIN {X 0,Y 473.348,Z 840.567,A -85,B 0,C 180,E1 21479.958,E2 21479.958} C_VEL
LIN {X 0,Y 475.857,Z 822.011,A -85,B 0,C 180,E1 21477.793,E2 21477.793} C_VEL
LIN {X 0,Y 477.656,Z 808.468,A -85,B 0,C 180,E1 21476.42,E2 21476.42} C_VEL
LIN {X 0,Y 479.935,Z 788.888,A -85,B 0,C 180,E1 21474.752,E2 21474.752} C_VEL
LIN {X 0,Y 482.019,Z 769.069,A -85,B 0,C 180,E1 21473.315,E2 21473.315} C_VEL
LIN {X 0,Y 484.227,Z 746.86,A -85,B 0,C 180,E1 21471.948,E2 21471.948} C_VEL
LIN {X 0,Y 486.041,Z 726.435,A -85,B 0,C 180,E1 21470.911,E2 21470.911} C_VEL
LIN {X 0,Y 487.805,Z 702.639,A -85,B 0,C 180,E1 21469.938,E2 21469.938} C_VEL
LIN {X 0,Y 489.161,Z 679.979,A -85,B 0,C 180,E1 21469.226,E2 21469.226} C_VEL
LIN {X 0,Y 490.137,Z 656.451,A -85,B 0,C 180,E1 21468.719,E2 21468.719} C_VEL
LIN {X 0,Y 493.497,Z 451.018,A -85,B 0,C 180,E1 21465.401,E2 21465.401} C_VEL
LIN {X 0,Y 495.297,Z 335.493,A -85,B 0,C 180,E1 21463.477,E2 21463.477} C_VEL
LIN {X 0,Y 493.393,Z 317.644,A -85,B 0,C 180,E1 21462.942,E2 21462.942} C_VEL
LIN {X 0,Y 494.678,Z 295.571,A -85,B 0,C 180,E1 21461.732,E2 21461.732} C_VEL
LIN {X 0,Y 484.894,Z 276.924,A -85,B 0,C 180,E1 21459.428,E2 21459.428} C_VEL
LIN {X 0,Y 475.645,Z 260.213,A -85,B 0,C 180,E1 21457.107,E2 21457.107} C_VEL
LIN {X 0,Y 470.065,Z 250.665,A -85,B 0,C 180,E1 21455.649,E2 21455.649} C_VEL
LIN {X 0,Y 467.988,Z 247.024,A -85,B 0,C 180,E1 21455.08,E2 21455.08} C_VEL
LIN {X 0,Y 465.291,Z 242.514,A -85,B 0,C 180,E1 21454.339,E2 21454.339} C_VEL
LIN {X 0,Y 464.97,Z 241.187,A -85,B 0,C 180,E1 21454.031,E2 21454.031} C_VEL
LIN {X 0,Y 465.008,Z 241.127,A -85,B 0,C 180,E1 21450.351,E2 21450.351} C_VEL
LIN {X 0,Y 464.97,Z 241.127,A -85,B 0,C 180,E1 21446.821,E2 21446.821} C_VEL
LIN {X 0,Y 464.952,Z 241.129,A -85,B 0,C 180,E1 21443.309,E2 21443.309} C_VEL
LIN {X 0,Y 464.977,Z 241.124,A -85,B 0,C 180,E1 21439.731,E2 21439.731} C_VEL
LIN {X 0,Y 465.013,Z 241.122,A -85,B 0,C 180,E1 21436.104,E2 21436.104} C_VEL
LIN {X 0,Y 464.98,Z 241.128,A -85,B 0,C 180,E1 21432.51,E2 21432.51} C_VEL
LIN {X 0,Y 464.965,Z 241.124,A -85,B 0,C 180,E1 21428.907,E2 21428.907} C_VEL
LIN {X 0,Y 464.98,Z 241.113,A -85,B 0,C 180,E1 21425.306,E2 21425.306} C_VEL
LIN {X 0,Y 465.014,Z 241.106,A -85,B 0,C 180,E1 21421.725,E2 21421.725} C_VEL
LIN {X 0,Y 464.994,Z 241.127,A -85,B 0,C 180,E1 21418.152,E2 21418.152} C_VEL
LIN {X 0,Y 464.976,Z 241.121,A -85,B 0,C 180,E1 21414.571,E2 21414.571} C_VEL
LIN {X 0,Y 464.99,Z 241.106,A -85,B 0,C 180,E1 21410.969,E2 21410.969} C_VEL
LIN {X 0,Y 465.014,Z 241.114,A -85,B 0,C 180,E1 21407.332,E2 21407.332} C_VEL
LIN {X 0,Y 465.013,Z 241.126,A -85,B 0,C 180,E1 21403.641,E2 21403.641} C_VEL
LIN {X 0,Y 464.993,Z 241.108,A -85,B 0,C 180,E1 21399.997,E2 21399.997} C_VEL
LIN {X 0,Y 464.99,Z 241.114,A -85,B 0,C 180,E1 21396.291,E2 21396.291} C_VEL
LIN {X 0,Y 465.008,Z 241.122,A -85,B 0,C 180,E1 21392.604,E2 21392.604} C_VEL
LIN {X 0,Y 465.013,Z 241.12,A -85,B 0,C 180,E1 21388.934,E2 21388.934} C_VEL
LIN {X 0,Y 465.009,Z 241.107,A -85,B 0,C 180,E1 21385.224,E2 21385.224} C_VEL
LIN {X 0,Y 465.007,Z 241.114,A -85,B 0,C 180,E1 21381.507,E2 21381.507} C_VEL
LIN {X 0,Y 465.003,Z 241.124,A -85,B 0,C 180,E1 21377.867,E2 21377.867} C_VEL
LIN {X 0,Y 465.01,Z 241.12,A -85,B 0,C 180,E1 21374.161,E2 21374.161} C_VEL
LIN {X 0,Y 465.005,Z 241.117,A -85,B 0,C 180,E1 21370.433,E2 21370.433} C_VEL
LIN {X 0,Y 464.998,Z 241.114,A -85,B 0,C 180,E1 21366.676,E2 21366.676} C_VEL
LIN {X 0,Y 465.006,Z 241.112,A -85,B 0,C 180,E1 21362.958,E2 21362.958} C_VEL
LIN {X 0,Y 465.01,Z 241.111,A -85,B 0,C 180,E1 21359.358,E2 21359.358} C_VEL
LIN {X 0,Y 465.01,Z 241.114,A -85,B 0,C 180,E1 21355.722,E2 21355.722} C_VEL
LIN {X 0,Y 464.985,Z 241.07,A -85,B 0,C 180,E1 21352.064,E2 21352.064} C_VEL
LIN {X 0,Y 465.007,Z 241.117,A -85,B 0,C 180,E1 21349.645,E2 21349.645} C_VEL
LIN {X 0,Y 465.454,Z 242.244,A -85,B 0,C 180,E1 21349.235,E2 21349.235} C_VEL
LIN {X 0,Y 466.015,Z 245.268,A -85,B 0,C 180,E1 21348.845,E2 21348.845} C_VEL
LIN {X 0,Y 465.489,Z 252.027,A -85,B 0,C 180,E1 21348.329,E2 21348.329} C_VEL
LIN {X 0,Y 465.082,Z 256.78,A -85,B 0,C 180,E1 21347.945,E2 21347.945} C_VEL
LIN {X 0,Y 465.635,Z 258.965,A -85,B 0,C 180,E1 21347.671,E2 21347.671} C_VEL
LIN {X 0,Y 473.064,Z 273.87,A -85,B 0,C 180,E1 21345.446,E2 21345.446} C_VEL
LIN {X 0,Y 481.304,Z 291.823,A -85,B 0,C 180,E1 21343.023,E2 21343.023} C_VEL
LIN {X 0,Y 477.698,Z 336.56,A -85,B 0,C 180,E1 21339.884,E2 21339.884} C_VEL
LIN {X 0,Y 473.774,Z 389.579,A -85,B 0,C 180,E1 21336.241,E2 21336.241} C_VEL
LIN {X 0,Y 472.65,Z 407.755,A -85,B 0,C 180,E1 21335.031,E2 21335.031} C_VEL
LIN {X 0,Y 476.141,Z 438.012,A -85,B 0,C 180,E1 21334.131,E2 21334.131} C_VEL
LIN {X 0,Y 471.485,Z 630.321,A -85,B 0,C 180,E1 21330.833,E2 21330.833} C_VEL
LIN {X 0,Y 470.556,Z 650.229,A -85,B 0,C 180,E1 21330.279,E2 21330.279} C_VEL
LIN {X 0,Y 469.392,Z 669.178,A -85,B 0,C 180,E1 21329.513,E2 21329.513} C_VEL
LIN {X 0,Y 467.984,Z 687.497,A -85,B 0,C 180,E1 21328.532,E2 21328.532} C_VEL
LIN {X 0,Y 466.422,Z 704.803,A -85,B 0,C 180,E1 21327.358,E2 21327.358} C_VEL
LIN {X 0,Y 464.81,Z 721.098,A -85,B 0,C 180,E1 21325.992,E2 21325.992} C_VEL
LIN {X 0,Y 463.148,Z 736.796,A -85,B 0,C 180,E1 21324.387,E2 21324.387} C_VEL
LIN {X 0,Y 461.617,Z 750.768,A -85,B 0,C 180,E1 21322.659,E2 21322.659} C_VEL
LIN {X 0,Y 460.221,Z 763.566,A -85,B 0,C 180,E1 21320.75,E2 21320.75} C_VEL
LIN {X 0,Y 459.041,Z 774.909,A -85,B 0,C 180,E1 21318.696,E2 21318.696} C_VEL
LIN {X 0,Y 458.125,Z 784.297,A -85,B 0,C 180,E1 21316.625,E2 21316.625} C_VEL
LIN {X 0,Y 457.444,Z 792.382,A -85,B 0,C 180,E1 21314.406,E2 21314.406} C_VEL
LIN {X 0,Y 456.982,Z 798.835,A -85,B 0,C 180,E1 21312.128,E2 21312.128} C_VEL
LIN {X 0,Y 456.689,Z 803.743,A -85,B 0,C 180,E1 21309.764,E2 21309.764} C_VEL
LIN {X 0,Y 456.543,Z 807.018,A -85,B 0,C 180,E1 21307.33,E2 21307.33} C_VEL
LIN {X 0,Y 456.493,Z 808.567,A -85,B 0,C 180,E1 21304.995,E2 21304.995} C_VEL
LIN {X 0,Y 456.507,Z 808.56,A -85,B 0,C 180,E1 21302.618,E2 21302.618} C_VEL
LIN {X 0,Y 456.601,Z 806.898,A -85,B 0,C 180,E1 21300.195,E2 21300.195} C_VEL
LIN {X 0,Y 456.79,Z 803.714,A -85,B 0,C 180,E1 21297.868,E2 21297.868} C_VEL
LIN {X 0,Y 457.147,Z 798.766,A -85,B 0,C 180,E1 21295.497,E2 21295.497} C_VEL
LIN {X 0,Y 457.672,Z 792.34,A -85,B 0,C 180,E1 21293.233,E2 21293.233} C_VEL
LIN {X 0,Y 458.478,Z 783.874,A -85,B 0,C 180,E1 21290.928,E2 21290.928} C_VEL
LIN {X 0,Y 459.557,Z 773.902,A -85,B 0,C 180,E1 21288.761,E2 21288.761} C_VEL
LIN {X 0,Y 460.855,Z 762.411,A -85,B 0,C 180,E1 21286.721,E2 21286.721} C_VEL
LIN {X 0,Y 462.324,Z 750.08,A -85,B 0,C 180,E1 21284.908,E2 21284.908} C_VEL
LIN {X 0,Y 463.991,Z 735.801,A -85,B 0,C 180,E1 21283.163,E2 21283.163} C_VEL
LIN {X 0,Y 465.674,Z 720.911,A -85,B 0,C 180,E1 21281.654,E2 21281.654} C_VEL
LIN {X 0,Y 467.378,Z 704.747,A -85,B 0,C 180,E1 21280.304,E2 21280.304} C_VEL
LIN {X 0,Y 469.049,Z 687.141,A -85,B 0,C 180,E1 21279.114,E2 21279.114} C_VEL
LIN {X 0,Y 470.517,Z 669.436,A -85,B 0,C 180,E1 21278.166,E2 21278.166} C_VEL
LIN {X 0,Y 471.779,Z 650.46,A -85,B 0,C 180,E1 21277.395,E2 21277.395} C_VEL
LIN {X 0,Y 472.783,Z 630.881,A -85,B 0,C 180,E1 21276.841,E2 21276.841} C_VEL
LIN {X 0,Y 478.017,Z 454.35,A -85,B 0,C 180,E1 21273.695,E2 21273.695} C_VEL
LIN {X 0,Y 478.387,Z 436.391,A -85,B 0,C 180,E1 21273.363,E2 21273.363} C_VEL
LIN {X 0,Y 474.468,Z 403.043,A -85,B 0,C 180,E1 21272.254,E2 21272.254} C_VEL
LIN {X 0,Y 479.044,Z 346.666,A -85,B 0,C 180,E1 21268.341,E2 21268.341} C_VEL
LIN {X 0,Y 483.8,Z 294.929,A -85,B 0,C 180,E1 21264.674,E2 21264.674} C_VEL
LIN {X 0,Y 475.543,Z 277.276,A -85,B 0,C 180,E1 21262.108,E2 21262.108} C_VEL
LIN {X 0,Y 467.476,Z 261.392,A -85,B 0,C 180,E1 21259.49,E2 21259.49} C_VEL
LIN {X 0,Y 461.929,Z 251.525,A -85,B 0,C 180,E1 21257.639,E2 21257.639} C_VEL
LIN {X 0,Y 459.991,Z 247.82,A -85,B 0,C 180,E1 21256.933,E2 21256.933} C_VEL
LIN {X 0,Y 457.513,Z 244.114,A -85,B 0,C 180,E1 21256.113,E2 21256.113} C_VEL
LIN {X 0,Y 457.024,Z 242.309,A -85,B 0,C 180,E1 21255.724,E2 21255.724} C_VEL
LIN {X 0,Y 457.008,Z 242.115,A -85,B 0,C 180,E1 21252.252,E2 21252.252} C_VEL
LIN {X 0,Y 457.053,Z 242.116,A -85,B 0,C 180,E1 21248.681,E2 21248.681} C_VEL
LIN {X 0,Y 457.009,Z 242.113,A -85,B 0,C 180,E1 21245.146,E2 21245.146} C_VEL
LIN {X 0,Y 456.995,Z 242.121,A -85,B 0,C 180,E1 21241.504,E2 21241.504} C_VEL
LIN {X 0,Y 457.006,Z 242.12,A -85,B 0,C 180,E1 21237.868,E2 21237.868} C_VEL
LIN {X 0,Y 457.046,Z 242.109,A -85,B 0,C 180,E1 21234.224,E2 21234.224} C_VEL
LIN {X 0,Y 457.018,Z 242.111,A -85,B 0,C 180,E1 21230.63,E2 21230.63} C_VEL
LIN {X 0,Y 456.992,Z 242.12,A -85,B 0,C 180,E1 21227.105,E2 21227.105} C_VEL
LIN {X 0,Y 457.006,Z 242.122,A -85,B 0,C 180,E1 21223.476,E2 21223.476} C_VEL
LIN {X 0,Y 457.05,Z 242.11,A -85,B 0,C 180,E1 21219.912,E2 21219.912} C_VEL
LIN {X 0,Y 457.007,Z 242.113,A -85,B 0,C 180,E1 21216.398,E2 21216.398} C_VEL
LIN {X 0,Y 456.995,Z 242.124,A -85,B 0,C 180,E1 21212.789,E2 21212.789} C_VEL
LIN {X 0,Y 457.015,Z 242.115,A -85,B 0,C 180,E1 21209.206,E2 21209.206} C_VEL
LIN {X 0,Y 457.046,Z 242.372,A -85,B 0,C 180,E1 21207.069,E2 21207.069} C_VEL
LIN {X 0,Y 457.506,Z 244.104,A -85,B 0,C 180,E1 21206.732,E2 21206.732} C_VEL
LIN {X 0,Y 459.461,Z 246.955,A -85,B 0,C 180,E1 21206.145,E2 21206.145} C_VEL
LIN {X 0,Y 460.264,Z 248.124,A -85,B 0,C 180,E1 21205.912,E2 21205.912} C_VEL
LIN {X 0,Y 462.566,Z 252.084,A -85,B 0,C 180,E1 21205.204,E2 21205.204} C_VEL
LIN {X 0,Y 468.585,Z 262.508,A -85,B 0,C 180,E1 21203.464,E2 21203.464} C_VEL
LIN {X 0,Y 477.258,Z 278.364,A -85,B 0,C 180,E1 21201.137,E2 21201.137} C_VEL
LIN {X 0,Y 486.739,Z 297.411,A -85,B 0,C 180,E1 21198.746,E2 21198.746} C_VEL
LIN {X 0,Y 487.441,Z 299.38,A -85,B 0,C 180,E1 21198.544,E2 21198.544} C_VEL
LIN {X 0,Y 486.148,Z 322.19,A -85,B 0,C 180,E1 21197.322,E2 21197.322} C_VEL
LIN {X 0,Y 487.91,Z 339.488,A -85,B 0,C 180,E1 21196.842,E2 21196.842} C_VEL
LIN {X 0,Y 484.775,Z 545.35,A -85,B 0,C 180,E1 21193.506,E2 21193.506} C_VEL
LIN {X 0,Y 482.933,Z 661.635,A -85,B 0,C 180,E1 21191.646,E2 21191.646} C_VEL
LIN {X 0,Y 481.832,Z 684.717,A -85,B 0,C 180,E1 21191.092,E2 21191.092} C_VEL
LIN {X 0,Y 480.481,Z 706.862,A -85,B 0,C 180,E1 21190.366,E2 21190.366} C_VEL
LIN {X 0,Y 478.754,Z 728.158,A -85,B 0,C 180,E1 21189.454,E2 21189.454} C_VEL
LIN {X 0,Y 476.816,Z 749.491,A -85,B 0,C 180,E1 21188.348,E2 21188.348} C_VEL
LIN {X 0,Y 474.629,Z 770.397,A -85,B 0,C 180,E1 21187.022,E2 21187.022} C_VEL
LIN {X 0,Y 472.304,Z 791.469,A -85,B 0,C 180,E1 21185.452,E2 21185.452} C_VEL
LIN {X 0,Y 470.022,Z 810.46,A -85,B 0,C 180,E1 21183.797,E2 21183.797} C_VEL
LIN {X 0,Y 467.612,Z 830.145,A -85,B 0,C 180,E1 21181.806,E2 21181.806} C_VEL
LIN {X 0,Y 465.85,Z 842.614,A -85,B 0,C 180,E1 21180.288,E2 21180.288} C_VEL
LIN {X 0,Y 463.541,Z 858.761,A -85,B 0,C 180,E1 21178.047,E2 21178.047} C_VEL
LIN {X 0,Y 461.521,Z 873.43,A -85,B 0,C 180,E1 21175.675,E2 21175.675} C_VEL
LIN {X 0,Y 459.752,Z 887.545,A -85,B 0,C 180,E1 21173.044,E2 21173.044} C_VEL
LIN {X 0,Y 458.454,Z 899.015,A -85,B 0,C 180,E1 21170.555,E2 21170.555} C_VEL
LIN {X 0,Y 457.385,Z 910.232,A -85,B 0,C 180,E1 21167.688,E2 21167.688} C_VEL
LIN {X 0,Y 456.708,Z 919.178,A -85,B 0,C 180,E1 21164.97,E2 21164.97} C_VEL
LIN {X 0,Y 456.266,Z 926.656,A -85,B 0,C 180,E1 21162.143,E2 21162.143} C_VEL
LIN {X 0,Y 456.047,Z 932.6,A -85,B 0,C 180,E1 21159.336,E2 21159.336} C_VEL
LIN {X 0,Y 455.947,Z 936.801,A -85,B 0,C 180,E1 21156.546,E2 21156.546} C_VEL
LIN {X 0,Y 455.913,Z 939.646,A -85,B 0,C 180,E1 21153.754,E2 21153.754} C_VEL
LIN {X 0,Y 455.91,Z 940.827,A -85,B 0,C 180,E1 21151.004,E2 21151.004} C_VEL
LIN {X 0,Y 455.899,Z 940.713,A -85,B 0,C 180,E1 21148.365,E2 21148.365} C_VEL
LIN {X 0,Y 455.907,Z 939.067,A -85,B 0,C 180,E1 21145.596,E2 21145.596} C_VEL
LIN {X 0,Y 455.95,Z 936.318,A -85,B 0,C 180,E1 21143.071,E2 21143.071} C_VEL
LIN {X 0,Y 456.062,Z 931.588,A -85,B 0,C 180,E1 21140.153,E2 21140.153} C_VEL
LIN {X 0,Y 456.293,Z 926.042,A -85,B 0,C 180,E1 21137.598,E2 21137.598} C_VEL
LIN {X 0,Y 456.786,Z 917.954,A -85,B 0,C 180,E1 21134.64,E2 21134.64} C_VEL
LIN {X 0,Y 457.466,Z 909.308,A -85,B 0,C 180,E1 21132.05,E2 21132.05} C_VEL
LIN {X 0,Y 458.565,Z 897.86,A -85,B 0,C 180,E1 21129.181,E2 21129.181} C_VEL
LIN {X 0,Y 459.991,Z 885.617,A -85,B 0,C 180,E1 21126.56,E2 21126.56} C_VEL
LIN {X 0,Y 461.731,Z 871.873,A -85,B 0,C 180,E1 21124.059,E2 21124.059} C_VEL
LIN {X 0,Y 463.786,Z 856.949,A -85,B 0,C 180,E1 21121.686,E2 21121.686} C_VEL
LIN {X 0,Y 466.005,Z 841.58,A -85,B 0,C 180,E1 21119.577,E2 21119.577} C_VEL
LIN {X 0,Y 467.772,Z 828.925,A -85,B 0,C 180,E1 21118.058,E2 21118.058} C_VEL
LIN {X 0,Y 470.23,Z 809.114,A -85,B 0,C 180,E1 21116.063,E2 21116.063} C_VEL
LIN {X 0,Y 472.713,Z 789.018,A -85,B 0,C 180,E1 21114.313,E2 21114.313} C_VEL
LIN {X 0,Y 474.962,Z 768.884,A -85,B 0,C 180,E1 21112.83,E2 21112.83} C_VEL
LIN {X 0,Y 477.194,Z 748.011,A -85,B 0,C 180,E1 21111.515,E2 21111.515} C_VEL
LIN {X 0,Y 479.094,Z 727.824,A -85,B 0,C 180,E1 21110.466,E2 21110.466} C_VEL
LIN {X 0,Y 480.95,Z 705.095,A -85,B 0,C 180,E1 21109.5,E2 21109.5} C_VEL
LIN {X 0,Y 482.332,Z 683.43,A -85,B 0,C 180,E1 21108.791,E2 21108.791} C_VEL
LIN {X 0,Y 483.509,Z 658.693,A -85,B 0,C 180,E1 21108.218,E2 21108.218} C_VEL
LIN {X 0,Y 487.089,Z 456.386,A -85,B 0,C 180,E1 21104.911,E2 21104.911} C_VEL
LIN {X 0,Y 489.11,Z 336.803,A -85,B 0,C 180,E1 21102.901,E2 21102.901} C_VEL
LIN {X 0,Y 487.195,Z 318.946,A -85,B 0,C 180,E1 21102.368,E2 21102.368} C_VEL
LIN {X 0,Y 488.416,Z 299.355,A -85,B 0,C 180,E1 21101.277,E2 21101.277} C_VEL
LIN {X 0,Y 477.899,Z 279.169,A -85,B 0,C 180,E1 21098.724,E2 21098.724} C_VEL
LIN {X 0,Y 467.608,Z 260.92,A -85,B 0,C 180,E1 21096.073,E2 21096.073} C_VEL
LIN {X 0,Y 461.997,Z 251.407,A -85,B 0,C 180,E1 21094.543,E2 21094.543} C_VEL
LIN {X 0,Y 459.603,Z 247.076,A -85,B 0,C 180,E1 21093.843,E2 21093.843} C_VEL
LIN {X 0,Y 457.475,Z 243.997,A -85,B 0,C 180,E1 21093.27,E2 21093.27} C_VEL
LIN {X 0,Y 457.069,Z 242.454,A -85,B 0,C 180,E1 21093.004,E2 21093.004} C_VEL
LIN {X 0,Y 457.022,Z 242.106,A -85,B 0,C 180,E1 21091.968,E2 21091.968} C_VEL
LIN {X 0,Y 457.07,Z 242.102,A -85,B 0,C 180,E1 21088.43,E2 21088.43} C_VEL
LIN {X 0,Y 457.031,Z 242.11,A -85,B 0,C 180,E1 21084.781,E2 21084.781} C_VEL
LIN {X 0,Y 457.017,Z 242.115,A -85,B 0,C 180,E1 21081.161,E2 21081.161} C_VEL
LIN {X 0,Y 457.026,Z 242.113,A -85,B 0,C 180,E1 21077.441,E2 21077.441} C_VEL
LIN {X 0,Y 457.071,Z 242.1,A -85,B 0,C 180,E1 21073.924,E2 21073.924} C_VEL
LIN {X 0,Y 457.061,Z 242.098,A -85,B 0,C 180,E1 21070.207,E2 21070.207} C_VEL
LIN {X 0,Y 457.032,Z 242.107,A -85,B 0,C 180,E1 21066.659,E2 21066.659} C_VEL
LIN {X 0,Y 457.032,Z 242.116,A -85,B 0,C 180,E1 21062.885,E2 21062.885} C_VEL
LIN {X 0,Y 457.053,Z 242.113,A -85,B 0,C 180,E1 21059.248,E2 21059.248} C_VEL
LIN {X 0,Y 457.074,Z 242.096,A -85,B 0,C 180,E1 21055.609,E2 21055.609} C_VEL
LIN {X 0,Y 457.064,Z 242.098,A -85,B 0,C 180,E1 21051.952,E2 21051.952} C_VEL
LIN {X 0,Y 457.047,Z 242.116,A -85,B 0,C 180,E1 21048.262,E2 21048.262} C_VEL
LIN {X 0,Y 457.046,Z 242.108,A -85,B 0,C 180,E1 21044.521,E2 21044.521} C_VEL
LIN {X 0,Y 457.064,Z 242.09,A -85,B 0,C 180,E1 21040.845,E2 21040.845} C_VEL
LIN {X 0,Y 457.074,Z 242.106,A -85,B 0,C 180,E1 21037.221,E2 21037.221} C_VEL
LIN {X 0,Y 457.073,Z 242.112,A -85,B 0,C 180,E1 21033.471,E2 21033.471} C_VEL
LIN {X 0,Y 457.059,Z 242.095,A -85,B 0,C 180,E1 21029.781,E2 21029.781} C_VEL
LIN {X 0,Y 457.059,Z 242.102,A -85,B 0,C 180,E1 21026.095,E2 21026.095} C_VEL
LIN {X 0,Y 457.072,Z 242.11,A -85,B 0,C 180,E1 21022.363,E2 21022.363} C_VEL
LIN {X 0,Y 457.07,Z 242.112,A -85,B 0,C 180,E1 21018.62,E2 21018.62} C_VEL
LIN {X 0,Y 457.065,Z 242.102,A -85,B 0,C 180,E1 21014.866,E2 21014.866} C_VEL
LIN {X 0,Y 457.076,Z 242.096,A -85,B 0,C 180,E1 21011.182,E2 21011.182} C_VEL
LIN {X 0,Y 457.066,Z 242.099,A -85,B 0,C 180,E1 21007.456,E2 21007.456} C_VEL
LIN {X 0,Y 457.071,Z 242.1,A -85,B 0,C 180,E1 21003.755,E2 21003.755} C_VEL
LIN {X 0,Y 457.063,Z 242.1,A -85,B 0,C 180,E1 21000.064,E2 21000.064} C_VEL
LIN {X 0,Y 457.053,Z 242.102,A -85,B 0,C 180,E1 20996.366,E2 20996.366} C_VEL
LIN {X 0,Y 457.063,Z 242.062,A -85,B 0,C 180,E1 20992.782,E2 20992.782} C_VEL
LIN {X 0,Y 457.075,Z 242.255,A -85,B 0,C 180,E1 20990.489,E2 20990.489} C_VEL
LIN {X 0,Y 457.401,Z 243.637,A -85,B 0,C 180,E1 20990.206,E2 20990.206} C_VEL
LIN {X 0,Y 459.73,Z 247.653,A -85,B 0,C 180,E1 20989.503,E2 20989.503} C_VEL
LIN {X 0,Y 465.635,Z 258.965,A -85,B 0,C 180,E1 20987.671,E2 20987.671} C_VEL
LIN {X 0,Y 467.385,Z 264.096,A -85,B 0,C 180,E1 20986.992,E2 20986.992} C_VEL
LIN {X 0,Y 468.399,Z 274.526,A -85,B 0,C 180,E1 20985.963,E2 20985.963} C_VEL
LIN {X 0,Y 469.586,Z 283.108,A -85,B 0,C 180,E1 20985.088,E2 20985.088} C_VEL
LIN {X 0,Y 470.36,Z 285.393,A -85,B 0,C 180,E1 20984.803,E2 20984.803} C_VEL
LIN {X 0,Y 474.905,Z 296.065,A -85,B 0,C 180,E1 20983.392,E2 20983.392} C_VEL
LIN {X 0,Y 470.227,Z 350.589,A -85,B 0,C 180,E1 20979.548,E2 20979.548} C_VEL
LIN {X 0,Y 465.987,Z 406.424,A -85,B 0,C 180,E1 20975.693,E2 20975.693} C_VEL
LIN {X 0,Y 469.696,Z 439.276,A -85,B 0,C 180,E1 20974.693,E2 20974.693} C_VEL
LIN {X 0,Y 464.762,Z 629.978,A -85,B 0,C 180,E1 20971.373,E2 20971.373} C_VEL
LIN {X 0,Y 463.809,Z 649.562,A -85,B 0,C 180,E1 20970.83,E2 20970.83} C_VEL
LIN {X 0,Y 462.584,Z 668.64,A -85,B 0,C 180,E1 20970.063,E2 20970.063} C_VEL
LIN {X 0,Y 461.084,Z 687.244,A -85,B 0,C 180,E1 20969.069,E2 20969.069} C_VEL
LIN {X 0,Y 459.424,Z 704.73,A -85,B 0,C 180,E1 20967.881,E2 20967.881} C_VEL
LIN {X 0,Y 457.7,Z 721.206,A -85,B 0,C 180,E1 20966.495,E2 20966.495} C_VEL
LIN {X 0,Y 455.955,Z 736.71,A -85,B 0,C 180,E1 20964.906,E2 20964.906} C_VEL
LIN {X 0,Y 454.235,Z 751.364,A -85,B 0,C 180,E1 20963.082,E2 20963.082} C_VEL
LIN {X 0,Y 452.788,Z 763.69,A -85,B 0,C 180,E1 20961.237,E2 20961.237} C_VEL
LIN {X 0,Y 451.493,Z 775.201,A -85,B 0,C 180,E1 20959.152,E2 20959.152} C_VEL
LIN {X 0,Y 450.415,Z 785.258,A -85,B 0,C 180,E1 20956.915,E2 20956.915} C_VEL
LIN {X 0,Y 449.664,Z 793.386,A -85,B 0,C 180,E1 20954.658,E2 20954.658} C_VEL
LIN {X 0,Y 449.144,Z 799.932,A -85,B 0,C 180,E1 20952.321,E2 20952.321} C_VEL
LIN {X 0,Y 448.818,Z 804.84,A -85,B 0,C 180,E1 20949.937,E2 20949.937} C_VEL
LIN {X 0,Y 448.65,Z 808.168,A -85,B 0,C 180,E1 20947.462,E2 20947.462} C_VEL
LIN {X 0,Y 448.591,Z 809.776,A -85,B 0,C 180,E1 20945.088,E2 20945.088} C_VEL
LIN {X 0,Y 448.605,Z 809.834,A -85,B 0,C 180,E1 20942.67,E2 20942.67} C_VEL
LIN {X 0,Y 448.708,Z 808.244,A -85,B 0,C 180,E1 20940.206,E2 20940.206} C_VEL
LIN {X 0,Y 448.932,Z 804.864,A -85,B 0,C 180,E1 20937.69,E2 20937.69} C_VEL
LIN {X 0,Y 449.336,Z 799.887,A -85,B 0,C 180,E1 20935.276,E2 20935.276} C_VEL
LIN {X 0,Y 449.935,Z 793.252,A -85,B 0,C 180,E1 20932.917,E2 20932.917} C_VEL
LIN {X 0,Y 450.812,Z 784.968,A -85,B 0,C 180,E1 20930.633,E2 20930.633} C_VEL
LIN {X 0,Y 451.994,Z 774.964,A -85,B 0,C 180,E1 20928.425,E2 20928.425} C_VEL
LIN {X 0,Y 453.404,Z 763.47,A -85,B 0,C 180,E1 20926.354,E2 20926.354} C_VEL
LIN {X 0,Y 455.054,Z 750.537,A -85,B 0,C 180,E1 20924.433,E2 20924.433} C_VEL
LIN {X 0,Y 456.784,Z 736.751,A -85,B 0,C 180,E1 20922.73,E2 20922.73} C_VEL
LIN {X 0,Y 458.651,Z 721.266,A -85,B 0,C 180,E1 20921.145,E2 20921.145} C_VEL
LIN {X 0,Y 460.489,Z 704.938,A -85,B 0,C 180,E1 20919.771,E2 20919.771} C_VEL
LIN {X 0,Y 462.208,Z 687.934,A -85,B 0,C 180,E1 20918.608,E2 20918.608} C_VEL
LIN {X 0,Y 463.78,Z 670.103,A -85,B 0,C 180,E1 20917.64,E2 20917.64} C_VEL
LIN {X 0,Y 465.13,Z 650.991,A -85,B 0,C 180,E1 20916.853,E2 20916.853} C_VEL
LIN {X 0,Y 466.195,Z 631.477,A -85,B 0,C 180,E1 20916.292,E2 20916.292} C_VEL
LIN {X 0,Y 471.456,Z 465.383,A -85,B 0,C 180,E1 20913.277,E2 20913.277} C_VEL
LIN {X 0,Y 472.194,Z 437.675,A -85,B 0,C 180,E1 20912.765,E2 20912.765} C_VEL
LIN {X 0,Y 468.079,Z 401.745,A -85,B 0,C 180,E1 20911.541,E2 20911.541} C_VEL
LIN {X 0,Y 472.98,Z 345.391,A -85,B 0,C 180,E1 20907.577,E2 20907.577} C_VEL
LIN {X 0,Y 477.512,Z 298.761,A -85,B 0,C 180,E1 20904.229,E2 20904.229} C_VEL
LIN {X 0,Y 469.709,Z 282.045,A -85,B 0,C 180,E1 20901.739,E2 20901.739} C_VEL
LIN {X 0,Y 462.096,Z 266.929,A -85,B 0,C 180,E1 20899.201,E2 20899.201} C_VEL
LIN {X 0,Y 456.636,Z 257.138,A -85,B 0,C 180,E1 20897.324,E2 20897.324} C_VEL
LIN {X 0,Y 454.379,Z 252.896,A -85,B 0,C 180,E1 20896.49,E2 20896.49} C_VEL
LIN {X 0,Y 452.368,Z 249.618,A -85,B 0,C 180,E1 20895.775,E2 20895.775} C_VEL
LIN {X 0,Y 451.453,Z 247.875,A -85,B 0,C 180,E1 20895.412,E2 20895.412} C_VEL
LIN {X 0,Y 449.493,Z 244.764,A -85,B 0,C 180,E1 20894.689,E2 20894.689} C_VEL
LIN {X 0,Y 449.08,Z 243.201,A -85,B 0,C 180,E1 20894.28,E2 20894.28} C_VEL
LIN {X 0,Y 449.105,Z 243.101,A -85,B 0,C 180,E1 20890.648,E2 20890.648} C_VEL
LIN {X 0,Y 449.085,Z 243.102,A -85,B 0,C 180,E1 20887.033,E2 20887.033} C_VEL
LIN {X 0,Y 449.056,Z 243.112,A -85,B 0,C 180,E1 20883.446,E2 20883.446} C_VEL
LIN {X 0,Y 449.058,Z 243.101,A -85,B 0,C 180,E1 20879.744,E2 20879.744} C_VEL
LIN {X 0,Y 449.095,Z 243.1,A -85,B 0,C 180,E1 20876.17,E2 20876.17} C_VEL
LIN {X 0,Y 449.102,Z 243.107,A -85,B 0,C 180,E1 20872.452,E2 20872.452} C_VEL
LIN {X 0,Y 449.063,Z 243.109,A -85,B 0,C 180,E1 20868.83,E2 20868.83} C_VEL
LIN {X 0,Y 449.052,Z 243.101,A -85,B 0,C 180,E1 20865.163,E2 20865.163} C_VEL
LIN {X 0,Y 449.076,Z 243.103,A -85,B 0,C 180,E1 20861.569,E2 20861.569} C_VEL
LIN {X 0,Y 449.124,Z 243.105,A -85,B 0,C 180,E1 20857.899,E2 20857.899} C_VEL
LIN {X 0,Y 449.075,Z 243.102,A -85,B 0,C 180,E1 20854.268,E2 20854.268} C_VEL
LIN {X 0,Y 449.055,Z 243.114,A -85,B 0,C 180,E1 20850.669,E2 20850.669} C_VEL
LIN {X 0,Y 449.088,Z 243.324,A -85,B 0,C 180,E1 20848.452,E2 20848.452} C_VEL
LIN {X 0,Y 449.644,Z 245.215,A -85,B 0,C 180,E1 20848.046,E2 20848.046} C_VEL
LIN {X 0,Y 452.308,Z 248.96,A -85,B 0,C 180,E1 20847.208,E2 20847.208} C_VEL
LIN {X 0,Y 454.435,Z 252.839,A -85,B 0,C 180,E1 20846.478,E2 20846.478} C_VEL
LIN {X 0,Y 455.607,Z 254.632,A -85,B 0,C 180,E1 20846.122,E2 20846.122} C_VEL
LIN {X 0,Y 461.825,Z 265.421,A -85,B 0,C 180,E1 20844.228,E2 20844.228} C_VEL
LIN {X 0,Y 468.396,Z 277.252,A -85,B 0,C 180,E1 20842.374,E2 20842.374} C_VEL
LIN {X 0,Y 476.969,Z 293.888,A -85,B 0,C 180,E1 20840.099,E2 20840.099} C_VEL
LIN {X 0,Y 481.161,Z 302.605,A -85,B 0,C 180,E1 20839.034,E2 20839.034} C_VEL
LIN {X 0,Y 479.884,Z 323.179,A -85,B 0,C 180,E1 20837.909,E2 20837.909} C_VEL
LIN {X 0,Y 481.624,Z 340.669,A -85,B 0,C 180,E1 20837.415,E2 20837.415} C_VEL
LIN {X 0,Y 478.242,Z 545.779,A -85,B 0,C 180,E1 20834.053,E2 20834.053} C_VEL
LIN {X 0,Y 476.309,Z 661.453,A -85,B 0,C 180,E1 20832.187,E2 20832.187} C_VEL
LIN {X 0,Y 475.143,Z 684.544,A -85,B 0,C 180,E1 20831.627,E2 20831.627} C_VEL
LIN {X 0,Y 473.738,Z 706.319,A -85,B 0,C 180,E1 20830.907,E2 20830.907} C_VEL
LIN {X 0,Y 471.895,Z 727.993,A -85,B 0,C 180,E1 20829.967,E2 20829.967} C_VEL
LIN {X 0,Y 469.823,Z 749.397,A -85,B 0,C 180,E1 20828.839,E2 20828.839} C_VEL
LIN {X 0,Y 467.503,Z 770.367,A -85,B 0,C 180,E1 20827.489,E2 20827.489} C_VEL
LIN {X 0,Y 464.897,Z 792.477,A -85,B 0,C 180,E1 20825.8,E2 20825.8} C_VEL
LIN {X 0,Y 462.429,Z 812.022,A -85,B 0,C 180,E1 20824.054,E2 20824.054} C_VEL
LIN {X 0,Y 459.989,Z 830.718,A -85,B 0,C 180,E1 20822.102,E2 20822.102} C_VEL
LIN {X 0,Y 457.632,Z 848.631,A -85,B 0,C 180,E1 20819.967,E2 20819.967} C_VEL
LIN {X 0,Y 455.798,Z 861.322,A -85,B 0,C 180,E1 20818.134,E2 20818.134} C_VEL
LIN {X 0,Y 453.706,Z 875.74,A -85,B 0,C 180,E1 20815.729,E2 20815.729} C_VEL
LIN {X 0,Y 451.937,Z 888.813,A -85,B 0,C 180,E1 20813.19,E2 20813.19} C_VEL
LIN {X 0,Y 450.521,Z 900.76,A -85,B 0,C 180,E1 20810.518,E2 20810.518} C_VEL
LIN {X 0,Y 449.446,Z 911.148,A -85,B 0,C 180,E1 20807.743,E2 20807.743} C_VEL
LIN {X 0,Y 448.707,Z 920.289,A -85,B 0,C 180,E1 20804.846,E2 20804.846} C_VEL
LIN {X 0,Y 448.288,Z 926.958,A -85,B 0,C 180,E1 20802.231,E2 20802.231} C_VEL
LIN {X 0,Y 448.054,Z 932.811,A -85,B 0,C 180,E1 20799.374,E2 20799.374} C_VEL
LIN {X 0,Y 447.948,Z 936.821,A -85,B 0,C 180,E1 20796.648,E2 20796.648} C_VEL
LIN {X 0,Y 447.913,Z 939.672,A -85,B 0,C 180,E1 20793.784,E2 20793.784} C_VEL
LIN {X 0,Y 447.911,Z 940.826,A -85,B 0,C 180,E1 20791.022,E2 20791.022} C_VEL
LIN {X 0,Y 447.899,Z 940.712,A -85,B 0,C 180,E1 20788.336,E2 20788.336} C_VEL
LIN {X 0,Y 447.907,Z 939.067,A -85,B 0,C 180,E1 20785.518,E2 20785.518} C_VEL
LIN {X 0,Y 447.955,Z 936.318,A -85,B 0,C 180,E1 20782.947,E2 20782.947} C_VEL
LIN {X 0,Y 448.077,Z 931.588,A -85,B 0,C 180,E1 20779.975,E2 20779.975} C_VEL
LIN {X 0,Y 448.336,Z 926.042,A -85,B 0,C 180,E1 20777.375,E2 20777.375} C_VEL
LIN {X 0,Y 448.872,Z 917.953,A -85,B 0,C 180,E1 20774.363,E2 20774.363} C_VEL
LIN {X 0,Y 449.617,Z 909.306,A -85,B 0,C 180,E1 20771.725,E2 20771.725} C_VEL
LIN {X 0,Y 450.754,Z 898.432,A -85,B 0,C 180,E1 20768.939,E2 20768.939} C_VEL
LIN {X 0,Y 452.186,Z 886.897,A -85,B 0,C 180,E1 20766.407,E2 20766.407} C_VEL
LIN {X 0,Y 454.028,Z 873.412,A -85,B 0,C 180,E1 20763.867,E2 20763.867} C_VEL
LIN {X 0,Y 456.195,Z 858.743,A -85,B 0,C 180,E1 20761.457,E2 20761.457} C_VEL
LIN {X 0,Y 458.15,Z 844.761,A -85,B 0,C 180,E1 20759.546,E2 20759.546} C_VEL
LIN {X 0,Y 460.478,Z 827.404,A -85,B 0,C 180,E1 20757.505,E2 20757.505} C_VEL
LIN {X 0,Y 463.031,Z 808.121,A -85,B 0,C 180,E1 20755.544,E2 20755.544} C_VEL
LIN {X 0,Y 465.601,Z 788.407,A -85,B 0,C 180,E1 20753.803,E2 20753.803} C_VEL
LIN {X 0,Y 468.058,Z 767.743,A -85,B 0,C 180,E1 20752.263,E2 20752.263} C_VEL
LIN {X 0,Y 470.554,Z 745.556,A -85,B 0,C 180,E1 20750.869,E2 20750.869} C_VEL
LIN {X 0,Y 472.506,Z 725.803,A -85,B 0,C 180,E1 20749.843,E2 20749.843} C_VEL
LIN {X 0,Y 474.484,Z 701.911,A -85,B 0,C 180,E1 20748.843,E2 20748.843} C_VEL
LIN {X 0,Y 476.029,Z 679.116,A -85,B 0,C 180,E1 20748.117,E2 20748.117} C_VEL
LIN {X 0,Y 477.081,Z 655.918,A -85,B 0,C 180,E1 20747.61,E2 20747.61} C_VEL
LIN {X 0,Y 481.012,Z 445.851,A -85,B 0,C 180,E1 20744.144,E2 20744.144} C_VEL
LIN {X 0,Y 482.968,Z 338.062,A -85,B 0,C 180,E1 20742.309,E2 20742.309} C_VEL
LIN {X 0,Y 481.074,Z 319.505,A -85,B 0,C 180,E1 20741.742,E2 20741.742} C_VEL
LIN {X 0,Y 482.165,Z 303.21,A -85,B 0,C 180,E1 20740.823,E2 20740.823} C_VEL
LIN {X 0,Y 472.671,Z 284.819,A -85,B 0,C 180,E1 20738.456,E2 20738.456} C_VEL
LIN {X 0,Y 462.734,Z 266.983,A -85,B 0,C 180,E1 20735.843,E2 20735.843} C_VEL
LIN {X 0,Y 454.437,Z 252.883,A -85,B 0,C 180,E1 20733.522,E2 20733.522} C_VEL
LIN {X 0,Y 452.407,Z 249.585,A -85,B 0,C 180,E1 20732.935,E2 20732.935} C_VEL
LIN {X 0,Y 451.677,Z 248.044,A -85,B 0,C 180,E1 20732.693,E2 20732.693} C_VEL
LIN {X 0,Y 449.593,Z 245.044,A -85,B 0,C 180,E1 20732.108,E2 20732.108} C_VEL
LIN {X 0,Y 449.139,Z 243.514,A -85,B 0,C 180,E1 20731.844,E2 20731.844} C_VEL
LIN {X 0,Y 449.069,Z 243.099,A -85,B 0,C 180,E1 20731.251,E2 20731.251} C_VEL
LIN {X 0,Y 449.073,Z 243.111,A -85,B 0,C 180,E1 20727.444,E2 20727.444} C_VEL
LIN {X 0,Y 449.092,Z 243.108,A -85,B 0,C 180,E1 20723.765,E2 20723.765} C_VEL
LIN {X 0,Y 449.132,Z 243.103,A -85,B 0,C 180,E1 20720.186,E2 20720.186} C_VEL
LIN {X 0,Y 449.113,Z 243.107,A -85,B 0,C 180,E1 20716.424,E2 20716.424} C_VEL
LIN {X 0,Y 449.089,Z 243.105,A -85,B 0,C 180,E1 20712.792,E2 20712.792} C_VEL
LIN {X 0,Y 449.09,Z 243.101,A -85,B 0,C 180,E1 20709.096,E2 20709.096} C_VEL
LIN {X 0,Y 449.116,Z 243.086,A -85,B 0,C 180,E1 20705.494,E2 20705.494} C_VEL
LIN {X 0,Y 449.136,Z 243.083,A -85,B 0,C 180,E1 20701.786,E2 20701.786} C_VEL
LIN {X 0,Y 449.121,Z 243.102,A -85,B 0,C 180,E1 20698.087,E2 20698.087} C_VEL
LIN {X 0,Y 449.104,Z 243.099,A -85,B 0,C 180,E1 20694.376,E2 20694.376} C_VEL
LIN {X 0,Y 449.101,Z 243.084,A -85,B 0,C 180,E1 20690.647,E2 20690.647} C_VEL
LIN {X 0,Y 449.124,Z 243.09,A -85,B 0,C 180,E1 20687.007,E2 20687.007} C_VEL
LIN {X 0,Y 449.136,Z 243.101,A -85,B 0,C 180,E1 20683.312,E2 20683.312} C_VEL
LIN {X 0,Y 449.135,Z 243.088,A -85,B 0,C 180,E1 20679.543,E2 20679.543} C_VEL
LIN {X 0,Y 449.121,Z 243.084,A -85,B 0,C 180,E1 20675.819,E2 20675.819} C_VEL
LIN {X 0,Y 449.117,Z 243.103,A -85,B 0,C 180,E1 20672.109,E2 20672.109} C_VEL
LIN {X 0,Y 449.124,Z 243.1,A -85,B 0,C 180,E1 20668.306,E2 20668.306} C_VEL
LIN {X 0,Y 449.131,Z 243.088,A -85,B 0,C 180,E1 20664.568,E2 20664.568} C_VEL
LIN {X 0,Y 449.127,Z 243.081,A -85,B 0,C 180,E1 20660.785,E2 20660.785} C_VEL
LIN {X 0,Y 449.13,Z 243.093,A -85,B 0,C 180,E1 20657.062,E2 20657.062} C_VEL
LIN {X 0,Y 449.132,Z 243.103,A -85,B 0,C 180,E1 20653.285,E2 20653.285} C_VEL
LIN {X 0,Y 449.129,Z 243.1,A -85,B 0,C 180,E1 20649.547,E2 20649.547} C_VEL
LIN {X 0,Y 449.133,Z 243.098,A -85,B 0,C 180,E1 20645.839,E2 20645.839} C_VEL
LIN {X 0,Y 449.125,Z 243.099,A -85,B 0,C 180,E1 20642.147,E2 20642.147} C_VEL
LIN {X 0,Y 449.118,Z 243.101,A -85,B 0,C 180,E1 20638.435,E2 20638.435} C_VEL
LIN {X 0,Y 449.127,Z 243.105,A -85,B 0,C 180,E1 20634.731,E2 20634.731} C_VEL
LIN {X 0,Y 449.148,Z 243.181,A -85,B 0,C 180,E1 20631.62,E2 20631.62} C_VEL
LIN {X 0,Y 449.582,Z 244.873,A -85,B 0,C 180,E1 20631.255,E2 20631.255} C_VEL
LIN {X 0,Y 451.767,Z 248.481,A -85,B 0,C 180,E1 20630.581,E2 20630.581} C_VEL
LIN {X 0,Y 453.979,Z 252.503,A -85,B 0,C 180,E1 20629.878,E2 20629.878} C_VEL
LIN {X 0,Y 462.868,Z 269.694,A -85,B 0,C 180,E1 20627.085,E2 20627.085} C_VEL
LIN {X 0,Y 470.36,Z 285.393,A -85,B 0,C 180,E1 20624.803,E2 20624.803} C_VEL
LIN {X 0,Y 471.257,Z 289.433,A -85,B 0,C 180,E1 20624.359,E2 20624.359} C_VEL
LIN {X 0,Y 470.946,Z 296.015,A -85,B 0,C 180,E1 20623.85,E2 20623.85} C_VEL
LIN {X 0,Y 467.004,Z 315.482,A -85,B 0,C 180,E1 20622.696,E2 20622.696} C_VEL
LIN {X 0,Y 466.895,Z 316.489,A -85,B 0,C 180,E1 20622.626,E2 20622.626} C_VEL
LIN {X 0,Y 461.941,Z 373.412,A -85,B 0,C 180,E1 20618.59,E2 20618.59} C_VEL
LIN {X 0,Y 459.459,Z 405.89,A -85,B 0,C 180,E1 20616.345,E2 20616.345} C_VEL
LIN {X 0,Y 463.291,Z 440.442,A -85,B 0,C 180,E1 20615.27,E2 20615.27} C_VEL
LIN {X 0,Y 458.079,Z 629.731,A -85,B 0,C 180,E1 20611.926,E2 20611.926} C_VEL
LIN {X 0,Y 457.096,Z 649.164,A -85,B 0,C 180,E1 20611.388,E2 20611.388} C_VEL
LIN {X 0,Y 455.817,Z 668.084,A -85,B 0,C 180,E1 20610.63,E2 20610.63} C_VEL
LIN {X 0,Y 454.316,Z 685.871,A -85,B 0,C 180,E1 20609.686,E2 20609.686} C_VEL
LIN {X 0,Y 452.639,Z 702.896,A -85,B 0,C 180,E1 20608.546,E2 20608.546} C_VEL
LIN {X 0,Y 450.846,Z 719.15,A -85,B 0,C 180,E1 20607.205,E2 20607.205} C_VEL
LIN {X 0,Y 449.02,Z 734.569,A -85,B 0,C 180,E1 20605.659,E2 20605.659} C_VEL
LIN {X 0,Y 447.229,Z 749.057,A -85,B 0,C 180,E1 20603.905,E2 20603.905} C_VEL
LIN {X 0,Y 445.584,Z 762.09,A -85,B 0,C 180,E1 20602.004,E2 20602.004} C_VEL
LIN {X 0,Y 444.199,Z 773.386,A -85,B 0,C 180,E1 20600.021,E2 20600.021} C_VEL
LIN {X 0,Y 443.027,Z 783.427,A -85,B 0,C 180,E1 20597.886,E2 20597.886} C_VEL
LIN {X 0,Y 442.096,Z 792.147,A -85,B 0,C 180,E1 20595.596,E2 20595.596} C_VEL
LIN {X 0,Y 441.436,Z 799.441,A -85,B 0,C 180,E1 20593.148,E2 20593.148} C_VEL
LIN {X 0,Y 441.005,Z 804.928,A -85,B 0,C 180,E1 20590.671,E2 20590.671} C_VEL
LIN {X 0,Y 440.782,Z 808.689,A -85,B 0,C 180,E1 20588.162,E2 20588.162} C_VEL
LIN {X 0,Y 440.69,Z 810.688,A -85,B 0,C 180,E1 20585.755,E2 20585.755} C_VEL
LIN {X 0,Y 440.692,Z 811.164,A -85,B 0,C 180,E1 20583.308,E2 20583.308} C_VEL
LIN {X 0,Y 440.775,Z 810.038,A -85,B 0,C 180,E1 20580.812,E2 20580.812} C_VEL
LIN {X 0,Y 440.979,Z 807.144,A -85,B 0,C 180,E1 20578.238,E2 20578.238} C_VEL
LIN {X 0,Y 441.366,Z 802.651,A -85,B 0,C 180,E1 20575.776,E2 20575.776} C_VEL
LIN {X 0,Y 441.975,Z 796.412,A -85,B 0,C 180,E1 20573.33,E2 20573.33} C_VEL
LIN {X 0,Y 442.865,Z 788.475,A -85,B 0,C 180,E1 20570.953,E2 20570.953} C_VEL
LIN {X 0,Y 444.045,Z 779.1,A -85,B 0,C 180,E1 20568.722,E2 20568.722} C_VEL
LIN {X 0,Y 445.456,Z 768.298,A -85,B 0,C 180,E1 20566.622,E2 20566.622} C_VEL
LIN {X 0,Y 447.195,Z 755.599,A -85,B 0,C 180,E1 20564.591,E2 20564.591} C_VEL
LIN {X 0,Y 449.055,Z 741.87,A -85,B 0,C 180,E1 20562.773,E2 20562.773} C_VEL
LIN {X 0,Y 450.931,Z 727.49,A -85,B 0,C 180,E1 20561.188,E2 20561.188} C_VEL
LIN {X 0,Y 452.923,Z 711.262,A -85,B 0,C 180,E1 20559.708,E2 20559.708} C_VEL
LIN {X 0,Y 454.891,Z 693.733,A -85,B 0,C 180,E1 20558.412,E2 20558.412} C_VEL
LIN {X 0,Y 456.651,Z 675.444,A -85,B 0,C 180,E1 20557.336,E2 20557.336} C_VEL
LIN {X 0,Y 458.187,Z 656.325,A -85,B 0,C 180,E1 20556.476,E2 20556.476} C_VEL
LIN {X 0,Y 459.4,Z 636.816,A -85,B 0,C 180,E1 20555.846,E2 20555.846} C_VEL
LIN {X 0,Y 460.465,Z 609.735,A -85,B 0,C 180,E1 20555.288,E2 20555.288} C_VEL
LIN {X 0,Y 466.052,Z 439.041,A -85,B 0,C 180,E1 20552.157,E2 20552.157} C_VEL
LIN {X 0,Y 461.77,Z 400.358,A -85,B 0,C 180,E1 20550.802,E2 20550.802} C_VEL
LIN {X 0,Y 467.124,Z 343.003,A -85,B 0,C 180,E1 20546.711,E2 20546.711} C_VEL
LIN {X 0,Y 471.246,Z 302.652,A -85,B 0,C 180,E1 20543.773,E2 20543.773} C_VEL
LIN {X 0,Y 463.919,Z 286.806,A -85,B 0,C 180,E1 20541.36,E2 20541.36} C_VEL
LIN {X 0,Y 456.762,Z 272.461,A -85,B 0,C 180,E1 20538.903,E2 20538.903} C_VEL
LIN {X 0,Y 451.378,Z 262.706,A -85,B 0,C 180,E1 20537.001,E2 20537.001} C_VEL
LIN {X 0,Y 449.133,Z 258.578,A -85,B 0,C 180,E1 20536.157,E2 20536.157} C_VEL
LIN {X 0,Y 446.62,Z 254.058,A -85,B 0,C 180,E1 20535.184,E2 20535.184} C_VEL
LIN {X 0,Y 444.438,Z 250.285,A -85,B 0,C 180,E1 20534.327,E2 20534.327} C_VEL
LIN {X 0,Y 443.457,Z 248.822,A -85,B 0,C 180,E1 20533.96,E2 20533.96} C_VEL
LIN {X 0,Y 441.591,Z 245.909,A -85,B 0,C 180,E1 20533.219,E2 20533.219} C_VEL
LIN {X 0,Y 441.205,Z 244.307,A -85,B 0,C 180,E1 20532.831,E2 20532.831} C_VEL
LIN {X 0,Y 441.144,Z 244.097,A -85,B 0,C 180,E1 20529.128,E2 20529.128} C_VEL
LIN {X 0,Y 441.116,Z 244.094,A -85,B 0,C 180,E1 20525.593,E2 20525.593} C_VEL
LIN {X 0,Y 441.12,Z 244.094,A -85,B 0,C 180,E1 20521.818,E2 20521.818} C_VEL
LIN {X 0,Y 441.165,Z 244.096,A -85,B 0,C 180,E1 20518.311,E2 20518.311} C_VEL
LIN {X 0,Y 441.158,Z 244.09,A -85,B 0,C 180,E1 20514.537,E2 20514.537} C_VEL
LIN {X 0,Y 441.118,Z 244.09,A -85,B 0,C 180,E1 20511.002,E2 20511.002} C_VEL
LIN {X 0,Y 441.116,Z 244.094,A -85,B 0,C 180,E1 20507.298,E2 20507.298} C_VEL
LIN {X 0,Y 441.144,Z 244.1,A -85,B 0,C 180,E1 20503.677,E2 20503.677} C_VEL
LIN {X 0,Y 441.17,Z 244.088,A -85,B 0,C 180,E1 20499.987,E2 20499.987} C_VEL
LIN {X 0,Y 441.125,Z 244.09,A -85,B 0,C 180,E1 20496.489,E2 20496.489} C_VEL
LIN {X 0,Y 441.118,Z 244.101,A -85,B 0,C 180,E1 20492.75,E2 20492.75} C_VEL
LIN {X 0,Y 441.187,Z 244.327,A -85,B 0,C 180,E1 20489.943,E2 20489.943} C_VEL
LIN {X 0,Y 441.696,Z 246.112,A -85,B 0,C 180,E1 20489.531,E2 20489.531} C_VEL
LIN {X 0,Y 443.808,Z 249.146,A -85,B 0,C 180,E1 20488.79,E2 20488.79} C_VEL
LIN {X 0,Y 444.534,Z 250.144,A -85,B 0,C 180,E1 20488.545,E2 20488.545} C_VEL
LIN {X 0,Y 446.575,Z 253.809,A -85,B 0,C 180,E1 20487.8,E2 20487.8} C_VEL
LIN {X 0,Y 447.702,Z 255.457,A -85,B 0,C 180,E1 20487.437,E2 20487.437} C_VEL
LIN {X 0,Y 450.286,Z 259.65,A -85,B 0,C 180,E1 20486.586,E2 20486.586} C_VEL
LIN {X 0,Y 458.385,Z 273.822,A -85,B 0,C 180,E1 20484.072,E2 20484.072} C_VEL
LIN {X 0,Y 466.571,Z 289.244,A -85,B 0,C 180,E1 20481.733,E2 20481.733} C_VEL
LIN {X 0,Y 474.935,Z 306.435,A -85,B 0,C 180,E1 20479.498,E2 20479.498} C_VEL
LIN {X 0,Y 473.689,Z 324.346,A -85,B 0,C 180,E1 20478.505,E2 20478.505} C_VEL
LIN {X 0,Y 475.385,Z 342.086,A -85,B 0,C 180,E1 20477.998,E2 20477.998} C_VEL
LIN {X 0,Y 471.742,Z 547.477,A -85,B 0,C 180,E1 20474.596,E2 20474.596} C_VEL
LIN {X 0,Y 469.734,Z 661.144,A -85,B 0,C 180,E1 20472.745,E2 20472.745} C_VEL
LIN {X 0,Y 468.503,Z 684.205,A -85,B 0,C 180,E1 20472.183,E2 20472.183} C_VEL
LIN {X 0,Y 466.959,Z 706.808,A -85,B 0,C 180,E1 20471.422,E2 20471.422} C_VEL
LIN {X 0,Y 465.053,Z 728.037,A -85,B 0,C 180,E1 20470.486,E2 20470.486} C_VEL
LIN {X 0,Y 462.872,Z 749.279,A -85,B 0,C 180,E1 20469.347,E2 20469.347} C_VEL
LIN {X 0,Y 460.487,Z 769.68,A -85,B 0,C 180,E1 20468.017,E2 20468.017} C_VEL
LIN {X 0,Y 457.719,Z 791.897,A -85,B 0,C 180,E1 20466.296,E2 20466.296} C_VEL
LIN {X 0,Y 455.213,Z 810.695,A -85,B 0,C 180,E1 20464.594,E2 20464.594} C_VEL
LIN {X 0,Y 452.623,Z 829.453,A -85,B 0,C 180,E1 20462.614,E2 20462.614} C_VEL
LIN {X 0,Y 450.115,Z 847.542,A -85,B 0,C 180,E1 20460.427,E2 20460.427} C_VEL
LIN {X 0,Y 447.841,Z 864.071,A -85,B 0,C 180,E1 20458.103,E2 20458.103} C_VEL
LIN {X 0,Y 446.327,Z 874.967,A -85,B 0,C 180,E1 20456.329,E2 20456.329} C_VEL
LIN {X 0,Y 444.296,Z 888.811,A -85,B 0,C 180,E1 20453.613,E2 20453.613} C_VEL
LIN {X 0,Y 442.759,Z 900.729,A -85,B 0,C 180,E1 20450.902,E2 20450.902} C_VEL
LIN {X 0,Y 441.592,Z 911.147,A -85,B 0,C 180,E1 20448.069,E2 20448.069} C_VEL
LIN {X 0,Y 440.787,Z 920.289,A -85,B 0,C 180,E1 20445.12,E2 20445.12} C_VEL
LIN {X 0,Y 440.326,Z 926.958,A -85,B 0,C 180,E1 20442.456,E2 20442.456} C_VEL
LIN {X 0,Y 440.066,Z 932.811,A -85,B 0,C 180,E1 20439.546,E2 20439.546} C_VEL
LIN {X 0,Y 439.951,Z 936.801,A -85,B 0,C 180,E1 20436.786,E2 20436.786} C_VEL
LIN {X 0,Y 439.912,Z 939.633,A -85,B 0,C 180,E1 20433.908,E2 20433.908} C_VEL
LIN {X 0,Y 439.911,Z 940.826,A -85,B 0,C 180,E1 20431.041,E2 20431.041} C_VEL
LIN {X 0,Y 439.901,Z 940.735,A -85,B 0,C 180,E1 20428.436,E2 20428.436} C_VEL
LIN {X 0,Y 439.907,Z 939.067,A -85,B 0,C 180,E1 20425.436,E2 20425.436} C_VEL
LIN {X 0,Y 439.963,Z 936.318,A -85,B 0,C 180,E1 20422.818,E2 20422.818} C_VEL
LIN {X 0,Y 440.096,Z 931.588,A -85,B 0,C 180,E1 20419.792,E2 20419.792} C_VEL
LIN {X 0,Y 440.383,Z 926.041,A -85,B 0,C 180,E1 20417.143,E2 20417.143} C_VEL
LIN {X 0,Y 440.967,Z 917.952,A -85,B 0,C 180,E1 20414.075,E2 20414.075} C_VEL
LIN {X 0,Y 441.783,Z 909.306,A -85,B 0,C 180,E1 20411.389,E2 20411.389} C_VEL
LIN {X 0,Y 443.025,Z 898.43,A -85,B 0,C 180,E1 20408.553,E2 20408.553} C_VEL
LIN {X 0,Y 444.597,Z 886.68,A -85,B 0,C 180,E1 20405.931,E2 20405.931} C_VEL
LIN {X 0,Y 446.555,Z 873.397,A -85,B 0,C 180,E1 20403.396,E2 20403.396} C_VEL
LIN {X 0,Y 448.087,Z 862.252,A -85,B 0,C 180,E1 20401.621,E2 20401.621} C_VEL
LIN {X 0,Y 450.441,Z 845.615,A -85,B 0,C 180,E1 20399.299,E2 20399.299} C_VEL
LIN {X 0,Y 452.833,Z 828.636,A -85,B 0,C 180,E1 20397.25,E2 20397.25} C_VEL
LIN {X 0,Y 455.663,Z 808.632,A -85,B 0,C 180,E1 20395.152,E2 20395.152} C_VEL
LIN {X 0,Y 458.263,Z 789.697,A -85,B 0,C 180,E1 20393.44,E2 20393.44} C_VEL
LIN {X 0,Y 460.856,Z 769.391,A -85,B 0,C 180,E1 20391.877,E2 20391.877} C_VEL
LIN {X 0,Y 463.331,Z 749.024,A -85,B 0,C 180,E1 20390.54,E2 20390.54} C_VEL
LIN {X 0,Y 465.565,Z 727.875,A -85,B 0,C 180,E1 20389.402,E2 20389.402} C_VEL
LIN {X 0,Y 467.581,Z 706.137,A -85,B 0,C 180,E1 20388.441,E2 20388.441} C_VEL
LIN {X 0,Y 469.175,Z 683.693,A -85,B 0,C 180,E1 20387.685,E2 20387.685} C_VEL
LIN {X 0,Y 470.506,Z 659.094,A -85,B 0,C 180,E1 20387.096,E2 20387.096} C_VEL
LIN {X 0,Y 474.707,Z 450.054,A -85,B 0,C 180,E1 20383.608,E2 20383.608} C_VEL
LIN {X 0,Y 476.89,Z 339.435,A -85,B 0,C 180,E1 20381.705,E2 20381.705} C_VEL
LIN {X 0,Y 475.006,Z 320.037,A -85,B 0,C 180,E1 20381.099,E2 20381.099} C_VEL
LIN {X 0,Y 475.948,Z 307.074,A -85,B 0,C 180,E1 20380.358,E2 20380.358} C_VEL
LIN {X 0,Y 466.973,Z 289.673,A -85,B 0,C 180,E1 20378.072,E2 20378.072} C_VEL
LIN {X 0,Y 457.558,Z 272.606,A -85,B 0,C 180,E1 20375.54,E2 20375.54} C_VEL
LIN {X 0,Y 449.506,Z 258.854,A -85,B 0,C 180,E1 20373.241,E2 20373.241} C_VEL
LIN {X 0,Y 446.553,Z 253.838,A -85,B 0,C 180,E1 20372.353,E2 20372.353} C_VEL
LIN {X 0,Y 444.26,Z 249.779,A -85,B 0,C 180,E1 20371.628,E2 20371.628} C_VEL
LIN {X 0,Y 441.796,Z 246.398,A -85,B 0,C 180,E1 20370.913,E2 20370.913} C_VEL
LIN {X 0,Y 441.226,Z 244.408,A -85,B 0,C 180,E1 20370.556,E2 20370.556} C_VEL
LIN {X 0,Y 441.149,Z 244.081,A -85,B 0,C 180,E1 20368.866,E2 20368.866} C_VEL
LIN {X 0,Y 441.135,Z 244.084,A -85,B 0,C 180,E1 20365.221,E2 20365.221} C_VEL
LIN {X 0,Y 441.141,Z 244.087,A -85,B 0,C 180,E1 20361.402,E2 20361.402} C_VEL
LIN {X 0,Y 441.172,Z 244.08,A -85,B 0,C 180,E1 20357.816,E2 20357.816} C_VEL
LIN {X 0,Y 441.199,Z 244.074,A -85,B 0,C 180,E1 20354.08,E2 20354.08} C_VEL
LIN {X 0,Y 441.174,Z 244.075,A -85,B 0,C 180,E1 20350.314,E2 20350.314} C_VEL
LIN {X 0,Y 441.15,Z 244.085,A -85,B 0,C 180,E1 20346.769,E2 20346.769} C_VEL
LIN {X 0,Y 441.156,Z 244.094,A -85,B 0,C 180,E1 20342.989,E2 20342.989} C_VEL
LIN {X 0,Y 441.183,Z 244.091,A -85,B 0,C 180,E1 20339.351,E2 20339.351} C_VEL
LIN {X 0,Y 441.196,Z 244.072,A -85,B 0,C 180,E1 20335.581,E2 20335.581} C_VEL
LIN {X 0,Y 441.196,Z 244.07,A -85,B 0,C 180,E1 20331.792,E2 20331.792} C_VEL
LIN {X 0,Y 441.182,Z 244.09,A -85,B 0,C 180,E1 20327.966,E2 20327.966} C_VEL
LIN {X 0,Y 441.17,Z 244.087,A -85,B 0,C 180,E1 20324.219,E2 20324.219} C_VEL
LIN {X 0,Y 441.171,Z 244.069,A -85,B 0,C 180,E1 20320.402,E2 20320.402} C_VEL
LIN {X 0,Y 441.186,Z 244.081,A -85,B 0,C 180,E1 20316.635,E2 20316.635} C_VEL
LIN {X 0,Y 441.198,Z 244.089,A -85,B 0,C 180,E1 20312.903,E2 20312.903} C_VEL
LIN {X 0,Y 441.195,Z 244.078,A -85,B 0,C 180,E1 20309.192,E2 20309.192} C_VEL
LIN {X 0,Y 441.19,Z 244.071,A -85,B 0,C 180,E1 20305.353,E2 20305.353} C_VEL
LIN {X 0,Y 441.187,Z 244.08,A -85,B 0,C 180,E1 20301.614,E2 20301.614} C_VEL
LIN {X 0,Y 441.187,Z 244.092,A -85,B 0,C 180,E1 20297.825,E2 20297.825} C_VEL
LIN {X 0,Y 441.193,Z 244.087,A -85,B 0,C 180,E1 20294.078,E2 20294.078} C_VEL
LIN {X 0,Y 441.194,Z 244.082,A -85,B 0,C 180,E1 20290.233,E2 20290.233} C_VEL
LIN {X 0,Y 441.183,Z 244.08,A -85,B 0,C 180,E1 20286.426,E2 20286.426} C_VEL
LIN {X 0,Y 441.182,Z 244.079,A -85,B 0,C 180,E1 20282.643,E2 20282.643} C_VEL
LIN {X 0,Y 441.192,Z 244.08,A -85,B 0,C 180,E1 20278.864,E2 20278.864} C_VEL
LIN {X 0,Y 441.197,Z 244.089,A -85,B 0,C 180,E1 20275.075,E2 20275.075} C_VEL
LIN {X 0,Y 441.22,Z 244.318,A -85,B 0,C 180,E1 20272.736,E2 20272.736} C_VEL
LIN {X 0,Y 442.244,Z 247.156,A -85,B 0,C 180,E1 20272.184,E2 20272.184} C_VEL
LIN {X 0,Y 443.933,Z 249.547,A -85,B 0,C 180,E1 20271.678,E2 20271.678} C_VEL
LIN {X 0,Y 445.836,Z 253.168,A -85,B 0,C 180,E1 20271.029,E2 20271.029} C_VEL
LIN {X 0,Y 453.831,Z 268.272,A -85,B 0,C 180,E1 20268.431,E2 20268.431} C_VEL
LIN {X 0,Y 461.87,Z 284.712,A -85,B 0,C 180,E1 20265.901,E2 20265.901} C_VEL
LIN {X 0,Y 468.512,Z 299.465,A -85,B 0,C 180,E1 20263.846,E2 20263.846} C_VEL
LIN {X 0,Y 466.895,Z 316.489,A -85,B 0,C 180,E1 20262.626,E2 20262.626} C_VEL
LIN {X 0,Y 465.481,Z 323.376,A -85,B 0,C 180,E1 20262.22,E2 20262.22} C_VEL
LIN {X 0,Y 458.87,Z 342.452,A -85,B 0,C 180,E1 20261.392,E2 20261.392} C_VEL
LIN {X 0,Y 457.751,Z 348.361,A -85,B 0,C 180,E1 20261.032,E2 20261.032} C_VEL
LIN {X 0,Y 453.022,Z 402.696,A -85,B 0,C 180,E1 20257.165,E2 20257.165} C_VEL
LIN {X 0,Y 453.077,Z 406.165,A -85,B 0,C 180,E1 20256.989,E2 20256.989} C_VEL
LIN {X 0,Y 456.932,Z 441.577,A -85,B 0,C 180,E1 20255.863,E2 20255.863} C_VEL
LIN {X 0,Y 451.453,Z 629.129,A -85,B 0,C 180,E1 20252.504,E2 20252.504} C_VEL
LIN {X 0,Y 450.428,Z 648.813,A -85,B 0,C 180,E1 20251.961,E2 20251.961} C_VEL
LIN {X 0,Y 449.098,Z 667.532,A -85,B 0,C 180,E1 20251.213,E2 20251.213} C_VEL
LIN {X 0,Y 447.516,Z 685.564,A -85,B 0,C 180,E1 20250.257,E2 20250.257} C_VEL
LIN {X 0,Y 445.677,Z 703.334,A -85,B 0,C 180,E1 20249.061,E2 20249.061} C_VEL
LIN {X 0,Y 443.739,Z 719.93,A -85,B 0,C 180,E1 20247.677,E2 20247.677} C_VEL
LIN {X 0,Y 441.8,Z 735.372,A -85,B 0,C 180,E1 20246.108,E2 20246.108} C_VEL
LIN {X 0,Y 439.892,Z 749.891,A -85,B 0,C 180,E1 20244.327,E2 20244.327} C_VEL
LIN {X 0,Y 438.129,Z 762.961,A -85,B 0,C 180,E1 20242.395,E2 20242.395} C_VEL
LIN {X 0,Y 436.637,Z 774.291,A -85,B 0,C 180,E1 20240.379,E2 20240.379} C_VEL
LIN {X 0,Y 435.368,Z 784.367,A -85,B 0,C 180,E1 20238.207,E2 20238.207} C_VEL
LIN {X 0,Y 434.353,Z 793.128,A -85,B 0,C 180,E1 20235.878,E2 20235.878} C_VEL
LIN {X 0,Y 433.625,Z 800.466,A -85,B 0,C 180,E1 20233.388,E2 20233.388} C_VEL
LIN {X 0,Y 433.149,Z 806,A -85,B 0,C 180,E1 20230.867,E2 20230.867} C_VEL
LIN {X 0,Y 432.888,Z 809.814,A -85,B 0,C 180,E1 20228.313,E2 20228.313} C_VEL
LIN {X 0,Y 432.785,Z 811.87,A -85,B 0,C 180,E1 20225.86,E2 20225.86} C_VEL
LIN {X 0,Y 432.787,Z 812.389,A -85,B 0,C 180,E1 20223.226,E2 20223.226} C_VEL
LIN {X 0,Y 432.882,Z 811.233,A -85,B 0,C 180,E1 20220.683,E2 20220.683} C_VEL
LIN {X 0,Y 433.116,Z 808.348,A -85,B 0,C 180,E1 20218.088,E2 20218.088} C_VEL
LIN {X 0,Y 433.546,Z 803.887,A -85,B 0,C 180,E1 20215.598,E2 20215.598} C_VEL
LIN {X 0,Y 434.228,Z 797.527,A -85,B 0,C 180,E1 20213.062,E2 20213.062} C_VEL
LIN {X 0,Y 435.2,Z 789.587,A -85,B 0,C 180,E1 20210.649,E2 20210.649} C_VEL
LIN {X 0,Y 436.528,Z 779.861,A -85,B 0,C 180,E1 20208.304,E2 20208.304} C_VEL
LIN {X 0,Y 438.079,Z 768.902,A -85,B 0,C 180,E1 20206.155,E2 20206.155} C_VEL
LIN {X 0,Y 439.871,Z 756.714,A -85,B 0,C 180,E1 20204.183,E2 20204.183} C_VEL
LIN {X 0,Y 441.819,Z 743.236,A -85,B 0,C 180,E1 20202.366,E2 20202.366} C_VEL
LIN {X 0,Y 443.869,Z 728.509,A -85,B 0,C 180,E1 20200.715,E2 20200.715} C_VEL
LIN {X 0,Y 445.987,Z 712.297,A -85,B 0,C 180,E1 20199.213,E2 20199.213} C_VEL
LIN {X 0,Y 448.035,Z 695.159,A -85,B 0,C 180,E1 20197.921,E2 20197.921} C_VEL
LIN {X 0,Y 449.919,Z 676.815,A -85,B 0,C 180,E1 20196.817,E2 20196.817} C_VEL
LIN {X 0,Y 451.575,Z 657.469,A -85,B 0,C 180,E1 20195.926,E2 20195.926} C_VEL
LIN {X 0,Y 452.886,Z 637.683,A -85,B 0,C 180,E1 20195.272,E2 20195.272} C_VEL
LIN {X 0,Y 453.983,Z 611.693,A -85,B 0,C 180,E1 20194.723,E2 20194.723} C_VEL
LIN {X 0,Y 459.982,Z 440.562,A -85,B 0,C 180,E1 20191.538,E2 20191.538} C_VEL
LIN {X 0,Y 455.513,Z 399.376,A -85,B 0,C 180,E1 20190.066,E2 20190.066} C_VEL
LIN {X 0,Y 461.253,Z 341.691,A -85,B 0,C 180,E1 20185.9,E2 20185.9} C_VEL
LIN {X 0,Y 465.013,Z 306.548,A -85,B 0,C 180,E1 20183.305,E2 20183.305} C_VEL
LIN {X 0,Y 457.511,Z 290.068,A -85,B 0,C 180,E1 20180.734,E2 20180.734} C_VEL
LIN {X 0,Y 449.514,Z 274.143,A -85,B 0,C 180,E1 20177.875,E2 20177.875} C_VEL
LIN {X 0,Y 444.297,Z 264.719,A -85,B 0,C 180,E1 20175.935,E2 20175.935} C_VEL
LIN {X 0,Y 441.447,Z 259.769,A -85,B 0,C 180,E1 20174.829,E2 20174.829} C_VEL
LIN {X 0,Y 439.059,Z 255.434,A -85,B 0,C 180,E1 20173.834,E2 20173.834} C_VEL
LIN {X 0,Y 436.891,Z 252.097,A -85,B 0,C 180,E1 20172.96,E2 20172.96} C_VEL
LIN {X 0,Y 436.152,Z 250.345,A -85,B 0,C 180,E1 20172.578,E2 20172.578} C_VEL
LIN {X 0,Y 433.88,Z 247.504,A -85,B 0,C 180,E1 20171.7,E2 20171.7} C_VEL
LIN {X 0,Y 433.25,Z 245.395,A -85,B 0,C 180,E1 20171.177,E2 20171.177} C_VEL
LIN {X 0,Y 433.185,Z 245.084,A -85,B 0,C 180,E1 20169.432,E2 20169.432} C_VEL
LIN {X 0,Y 433.178,Z 245.083,A -85,B 0,C 180,E1 20165.696,E2 20165.696} C_VEL
LIN {X 0,Y 433.189,Z 245.08,A -85,B 0,C 180,E1 20161.984,E2 20161.984} C_VEL
LIN {X 0,Y 433.232,Z 245.082,A -85,B 0,C 180,E1 20158.413,E2 20158.413} C_VEL
LIN {X 0,Y 433.215,Z 245.079,A -85,B 0,C 180,E1 20154.57,E2 20154.57} C_VEL
LIN {X 0,Y 433.18,Z 245.078,A -85,B 0,C 180,E1 20150.969,E2 20150.969} C_VEL
LIN {X 0,Y 433.176,Z 245.083,A -85,B 0,C 180,E1 20147.197,E2 20147.197} C_VEL
LIN {X 0,Y 433.193,Z 245.089,A -85,B 0,C 180,E1 20143.507,E2 20143.507} C_VEL
LIN {X 0,Y 433.228,Z 245.075,A -85,B 0,C 180,E1 20139.886,E2 20139.886} C_VEL
LIN {X 0,Y 433.196,Z 245.078,A -85,B 0,C 180,E1 20136.321,E2 20136.321} C_VEL
LIN {X 0,Y 433.18,Z 245.088,A -85,B 0,C 180,E1 20132.656,E2 20132.656} C_VEL
LIN {X 0,Y 433.261,Z 245.297,A -85,B 0,C 180,E1 20131.615,E2 20131.615} C_VEL
LIN {X 0,Y 433.736,Z 247.15,A -85,B 0,C 180,E1 20131.158,E2 20131.158} C_VEL
LIN {X 0,Y 435.975,Z 250.22,A -85,B 0,C 180,E1 20130.305,E2 20130.305} C_VEL
LIN {X 0,Y 436.714,Z 251.054,A -85,B 0,C 180,E1 20130.058,E2 20130.058} C_VEL
LIN {X 0,Y 438.55,Z 254.701,A -85,B 0,C 180,E1 20129.289,E2 20129.289} C_VEL
LIN {X 0,Y 440.014,Z 256.591,A -85,B 0,C 180,E1 20128.795,E2 20128.795} C_VEL
LIN {X 0,Y 442.647,Z 260.846,A -85,B 0,C 180,E1 20127.862,E2 20127.862} C_VEL
LIN {X 0,Y 449.39,Z 272.679,A -85,B 0,C 180,E1 20125.588,E2 20125.588} C_VEL
LIN {X 0,Y 456.063,Z 284.66,A -85,B 0,C 180,E1 20123.549,E2 20123.549} C_VEL
LIN {X 0,Y 464.019,Z 300.347,A -85,B 0,C 180,E1 20121.26,E2 20121.26} C_VEL
LIN {X 0,Y 468.703,Z 310.221,A -85,B 0,C 180,E1 20119.978,E2 20119.978} C_VEL
LIN {X 0,Y 467.579,Z 325.338,A -85,B 0,C 180,E1 20119.13,E2 20119.13} C_VEL
LIN {X 0,Y 469.229,Z 343.354,A -85,B 0,C 180,E1 20118.604,E2 20118.604} C_VEL
LIN {X 0,Y 465.312,Z 548.156,A -85,B 0,C 180,E1 20115.173,E2 20115.173} C_VEL
LIN {X 0,Y 463.195,Z 661.131,A -85,B 0,C 180,E1 20113.315,E2 20113.315} C_VEL
LIN {X 0,Y 461.891,Z 684.15,A -85,B 0,C 180,E1 20112.745,E2 20112.745} C_VEL
LIN {X 0,Y 460.295,Z 706.345,A -85,B 0,C 180,E1 20111.991,E2 20111.991} C_VEL
LIN {X 0,Y 458.297,Z 727.569,A -85,B 0,C 180,E1 20111.045,E2 20111.045} C_VEL
LIN {X 0,Y 455.963,Z 749.153,A -85,B 0,C 180,E1 20109.87,E2 20109.87} C_VEL
LIN {X 0,Y 453.458,Z 769.483,A -85,B 0,C 180,E1 20108.526,E2 20108.526} C_VEL
LIN {X 0,Y 450.572,Z 791.319,A -85,B 0,C 180,E1 20106.807,E2 20106.807} C_VEL
LIN {X 0,Y 447.845,Z 810.812,A -85,B 0,C 180,E1 20105.012,E2 20105.012} C_VEL
LIN {X 0,Y 445.088,Z 829.571,A -85,B 0,C 180,E1 20102.983,E2 20102.983} C_VEL
LIN {X 0,Y 442.413,Z 847.834,A -85,B 0,C 180,E1 20100.713,E2 20100.713} C_VEL
LIN {X 0,Y 440.147,Z 863.5,A -85,B 0,C 180,E1 20098.463,E2 20098.463} C_VEL
LIN {X 0,Y 437.943,Z 879.309,A -85,B 0,C 180,E1 20095.851,E2 20095.851} C_VEL
LIN {X 0,Y 436.669,Z 888.773,A -85,B 0,C 180,E1 20094.051,E2 20094.051} C_VEL
LIN {X 0,Y 435.087,Z 900.156,A -85,B 0,C 180,E1 20091.43,E2 20091.43} C_VEL
LIN {X 0,Y 433.799,Z 910.687,A -85,B 0,C 180,E1 20088.545,E2 20088.545} C_VEL
LIN {X 0,Y 432.927,Z 919.724,A -85,B 0,C 180,E1 20085.619,E2 20085.619} C_VEL
LIN {X 0,Y 432.39,Z 926.654,A -85,B 0,C 180,E1 20082.824,E2 20082.824} C_VEL
LIN {X 0,Y 432.082,Z 932.601,A -85,B 0,C 180,E1 20079.858,E2 20079.858} C_VEL
LIN {X 0,Y 431.956,Z 936.801,A -85,B 0,C 180,E1 20076.912,E2 20076.912} C_VEL
LIN {X 0,Y 431.912,Z 939.633,A -85,B 0,C 180,E1 20073.981,E2 20073.981} C_VEL
LIN {X 0,Y 431.911,Z 940.826,A -85,B 0,C 180,E1 20071.06,E2 20071.06} C_VEL
LIN {X 0,Y 431.9,Z 940.735,A -85,B 0,C 180,E1 20068.407,E2 20068.407} C_VEL
LIN {X 0,Y 431.907,Z 939.067,A -85,B 0,C 180,E1 20065.351,E2 20065.351} C_VEL
LIN {X 0,Y 431.97,Z 936.318,A -85,B 0,C 180,E1 20062.685,E2 20062.685} C_VEL
LIN {X 0,Y 432.128,Z 931.462,A -85,B 0,C 180,E1 20059.535,E2 20059.535} C_VEL
LIN {X 0,Y 432.455,Z 925.738,A -85,B 0,C 180,E1 20056.767,E2 20056.767} C_VEL
LIN {X 0,Y 433.11,Z 917.546,A -85,B 0,C 180,E1 20053.64,E2 20053.64} C_VEL
LIN {X 0,Y 434.023,Z 908.846,A -85,B 0,C 180,E1 20050.904,E2 20050.904} C_VEL
LIN {X 0,Y 435.397,Z 897.856,A -85,B 0,C 180,E1 20048.017,E2 20048.017} C_VEL
LIN {X 0,Y 436.859,Z 887.439,A -85,B 0,C 180,E1 20045.67,E2 20045.67} C_VEL
LIN {X 0,Y 438.904,Z 872.524,A -85,B 0,C 180,E1 20042.965,E2 20042.965} C_VEL
LIN {X 0,Y 441.21,Z 856.75,A -85,B 0,C 180,E1 20040.483,E2 20040.483} C_VEL
LIN {X 0,Y 443.719,Z 839.661,A -85,B 0,C 180,E1 20038.177,E2 20038.177} C_VEL
LIN {X 0,Y 446.479,Z 821.476,A -85,B 0,C 180,E1 20036.03,E2 20036.03} C_VEL
LIN {X 0,Y 449.169,Z 803.143,A -85,B 0,C 180,E1 20034.165,E2 20034.165} C_VEL
LIN {X 0,Y 452.167,Z 782.205,A -85,B 0,C 180,E1 20032.338,E2 20032.338} C_VEL
LIN {X 0,Y 454.815,Z 762.615,A -85,B 0,C 180,E1 20030.88,E2 20030.88} C_VEL
LIN {X 0,Y 457.305,Z 741.843,A -85,B 0,C 180,E1 20029.587,E2 20029.587} C_VEL
LIN {X 0,Y 459.64,Z 720.378,A -85,B 0,C 180,E1 20028.476,E2 20028.476} C_VEL
LIN {X 0,Y 461.623,Z 698.02,A -85,B 0,C 180,E1 20027.574,E2 20027.574} C_VEL
LIN {X 0,Y 463.307,Z 674.401,A -85,B 0,C 180,E1 20026.854,E2 20026.854} C_VEL
LIN {X 0,Y 464.296,Z 652.454,A -85,B 0,C 180,E1 20026.387,E2 20026.387} C_VEL
LIN {X 0,Y 468.657,Z 444.389,A -85,B 0,C 180,E1 20022.888,E2 20022.888} C_VEL
LIN {X 0,Y 470.835,Z 340.645,A -85,B 0,C 180,E1 20021.082,E2 20021.082} C_VEL
LIN {X 0,Y 468.984,Z 320.463,A -85,B 0,C 180,E1 20020.436,E2 20020.436} C_VEL
LIN {X 0,Y 469.641,Z 310.688,A -85,B 0,C 180,E1 20019.853,E2 20019.853} C_VEL
LIN {X 0,Y 459.557,Z 291.272,A -85,B 0,C 180,E1 20017.218,E2 20017.218} C_VEL
LIN {X 0,Y 450.315,Z 274.549,A -85,B 0,C 180,E1 20014.64,E2 20014.64} C_VEL
LIN {X 0,Y 444.192,Z 264.265,A -85,B 0,C 180,E1 20012.853,E2 20012.853} C_VEL
LIN {X 0,Y 441.021,Z 258.96,A -85,B 0,C 180,E1 20011.887,E2 20011.887} C_VEL
LIN {X 0,Y 438.736,Z 255.008,A -85,B 0,C 180,E1 20011.153,E2 20011.153} C_VEL
LIN {X 0,Y 436.485,Z 251.129,A -85,B 0,C 180,E1 20010.414,E2 20010.414} C_VEL
LIN {X 0,Y 435.706,Z 249.935,A -85,B 0,C 180,E1 20010.17,E2 20010.17} C_VEL
LIN {X 0,Y 433.73,Z 247.123,A -85,B 0,C 180,E1 20009.56,E2 20009.56} C_VEL
LIN {X 0,Y 433.241,Z 245.393,A -85,B 0,C 180,E1 20009.223,E2 20009.223} C_VEL
LIN {X 0,Y 433.211,Z 245.078,A -85,B 0,C 180,E1 20007.873,E2 20007.873} C_VEL
LIN {X 0,Y 433.242,Z 245.083,A -85,B 0,C 180,E1 20004.11,E2 20004.11} C_VEL
LIN {X 0,Y 433.242,Z 245.084,A -85,B 0,C 180,E1 20000.395,E2 20000.395} C_VEL
LIN {X 0,Y 433.22,Z 245.085,A -85,B 0,C 180,E1 19996.63,E2 19996.63} C_VEL
LIN {X 0,Y 433.207,Z 245.083,A -85,B 0,C 180,E1 19992.937,E2 19992.937} C_VEL
LIN {X 0,Y 433.214,Z 245.075,A -85,B 0,C 180,E1 19989.164,E2 19989.164} C_VEL
LIN {X 0,Y 433.242,Z 245.061,A -85,B 0,C 180,E1 19985.563,E2 19985.563} C_VEL
LIN {X 0,Y 433.258,Z 245.058,A -85,B 0,C 180,E1 19981.72,E2 19981.72} C_VEL
LIN {X 0,Y 433.246,Z 245.077,A -85,B 0,C 180,E1 19978.017,E2 19978.017} C_VEL
LIN {X 0,Y 433.229,Z 245.077,A -85,B 0,C 180,E1 19974.305,E2 19974.305} C_VEL
LIN {X 0,Y 433.224,Z 245.061,A -85,B 0,C 180,E1 19970.569,E2 19970.569} C_VEL
LIN {X 0,Y 433.236,Z 245.065,A -85,B 0,C 180,E1 19966.793,E2 19966.793} C_VEL
LIN {X 0,Y 433.257,Z 245.078,A -85,B 0,C 180,E1 19963.096,E2 19963.096} C_VEL
LIN {X 0,Y 433.259,Z 245.068,A -85,B 0,C 180,E1 19959.324,E2 19959.324} C_VEL
LIN {X 0,Y 433.25,Z 245.058,A -85,B 0,C 180,E1 19955.601,E2 19955.601} C_VEL
LIN {X 0,Y 433.246,Z 245.07,A -85,B 0,C 180,E1 19951.765,E2 19951.765} C_VEL
LIN {X 0,Y 433.244,Z 245.08,A -85,B 0,C 180,E1 19947.941,E2 19947.941} C_VEL
LIN {X 0,Y 433.245,Z 245.071,A -85,B 0,C 180,E1 19944.102,E2 19944.102} C_VEL
LIN {X 0,Y 433.253,Z 245.056,A -85,B 0,C 180,E1 19940.265,E2 19940.265} C_VEL
LIN {X 0,Y 433.253,Z 245.062,A -85,B 0,C 180,E1 19936.441,E2 19936.441} C_VEL
LIN {X 0,Y 433.25,Z 245.072,A -85,B 0,C 180,E1 19932.593,E2 19932.593} C_VEL
LIN {X 0,Y 433.247,Z 245.077,A -85,B 0,C 180,E1 19928.714,E2 19928.714} C_VEL
LIN {X 0,Y 433.251,Z 245.079,A -85,B 0,C 180,E1 19924.914,E2 19924.914} C_VEL
LIN {X 0,Y 433.259,Z 245.077,A -85,B 0,C 180,E1 19921.112,E2 19921.112} C_VEL
LIN {X 0,Y 433.259,Z 245.071,A -85,B 0,C 180,E1 19917.318,E2 19917.318} C_VEL
LIN {X 0,Y 433.277,Z 245.31,A -85,B 0,C 180,E1 19913.961,E2 19913.961} C_VEL
LIN {X 0,Y 434.579,Z 248.548,A -85,B 0,C 180,E1 19913.313,E2 19913.313} C_VEL
LIN {X 0,Y 436.178,Z 250.954,A -85,B 0,C 180,E1 19912.794,E2 19912.794} C_VEL
LIN {X 0,Y 439.181,Z 256.502,A -85,B 0,C 180,E1 19911.743,E2 19911.743} C_VEL
LIN {X 0,Y 444.563,Z 266.522,A -85,B 0,C 180,E1 19909.932,E2 19909.932} C_VEL
LIN {X 0,Y 451.944,Z 280.869,A -85,B 0,C 180,E1 19907.54,E2 19907.54} C_VEL
LIN {X 0,Y 460.589,Z 299.577,A -85,B 0,C 180,E1 19904.779,E2 19904.779} C_VEL
LIN {X 0,Y 462.107,Z 303.289,A -85,B 0,C 180,E1 19904.281,E2 19904.281} C_VEL
LIN {X 0,Y 457.751,Z 348.361,A -85,B 0,C 180,E1 19901.032,E2 19901.032} C_VEL
LIN {X 0,Y 456.358,Z 355.264,A -85,B 0,C 180,E1 19900.622,E2 19900.622} C_VEL
LIN {X 0,Y 449.69,Z 374.341,A -85,B 0,C 180,E1 19899.782,E2 19899.782} C_VEL
LIN {X 0,Y 448.535,Z 380.257,A -85,B 0,C 180,E1 19899.42,E2 19899.42} C_VEL
LIN {X 0,Y 446.527,Z 404.338,A -85,B 0,C 180,E1 19897.722,E2 19897.722} C_VEL
LIN {X 0,Y 450.616,Z 442.779,A -85,B 0,C 180,E1 19896.471,E2 19896.471} C_VEL
LIN {X 0,Y 444.89,Z 628.222,A -85,B 0,C 180,E1 19893.105,E2 19893.105} C_VEL
LIN {X 0,Y 443.814,Z 648.332,A -85,B 0,C 180,E1 19892.556,E2 19892.556} C_VEL
LIN {X 0,Y 442.377,Z 667.669,A -85,B 0,C 180,E1 19891.782,E2 19891.782} C_VEL
LIN {X 0,Y 440.658,Z 686.344,A -85,B 0,C 180,E1 19890.781,E2 19890.781} C_VEL
LIN {X 0,Y 438.705,Z 704.19,A -85,B 0,C 180,E1 19889.562,E2 19889.562} C_VEL
LIN {X 0,Y 436.664,Z 720.706,A -85,B 0,C 180,E1 19888.164,E2 19888.164} C_VEL
LIN {X 0,Y 434.608,Z 736.168,A -85,B 0,C 180,E1 19886.572,E2 19886.572} C_VEL
LIN {X 0,Y 432.578,Z 750.72,A -85,B 0,C 180,E1 19884.763,E2 19884.763} C_VEL
LIN {X 0,Y 430.696,Z 763.829,A -85,B 0,C 180,E1 19882.8,E2 19882.8} C_VEL
LIN {X 0,Y 429.092,Z 775.201,A -85,B 0,C 180,E1 19880.749,E2 19880.749} C_VEL
LIN {X 0,Y 427.726,Z 785.315,A -85,B 0,C 180,E1 19878.541,E2 19878.541} C_VEL
LIN {X 0,Y 426.622,Z 794.117,A -85,B 0,C 180,E1 19876.171,E2 19876.171} C_VEL
LIN {X 0,Y 425.821,Z 801.498,A -85,B 0,C 180,E1 19873.636,E2 19873.636} C_VEL
LIN {X 0,Y 425.298,Z 807.075,A -85,B 0,C 180,E1 19871.071,E2 19871.071} C_VEL
LIN {X 0,Y 425,Z 810.939,A -85,B 0,C 180,E1 19868.471,E2 19868.471} C_VEL
LIN {X 0,Y 424.881,Z 813.126,A -85,B 0,C 180,E1 19865.83,E2 19865.83} C_VEL
LIN {X 0,Y 424.882,Z 813.631,A -85,B 0,C 180,E1 19863.292,E2 19863.292} C_VEL
LIN {X 0,Y 424.986,Z 812.545,A -85,B 0,C 180,E1 19860.704,E2 19860.704} C_VEL
LIN {X 0,Y 425.237,Z 809.737,A -85,B 0,C 180,E1 19858.061,E2 19858.061} C_VEL
LIN {X 0,Y 425.7,Z 805.36,A -85,B 0,C 180,E1 19855.527,E2 19855.527} C_VEL
LIN {X 0,Y 426.432,Z 799.1,A -85,B 0,C 180,E1 19852.947,E2 19852.947} C_VEL
LIN {X 0,Y 427.469,Z 791.277,A -85,B 0,C 180,E1 19850.492,E2 19850.492} C_VEL
LIN {X 0,Y 428.83,Z 782.004,A -85,B 0,C 180,E1 19848.179,E2 19848.179} C_VEL
LIN {X 0,Y 430.519,Z 770.871,A -85,B 0,C 180,E1 19845.922,E2 19845.922} C_VEL
LIN {X 0,Y 432.486,Z 758.353,A -85,B 0,C 180,E1 19843.84,E2 19843.84} C_VEL
LIN {X 0,Y 434.648,Z 744.361,A -85,B 0,C 180,E1 19841.914,E2 19841.914} C_VEL
LIN {X 0,Y 436.94,Z 728.903,A -85,B 0,C 180,E1 19840.158,E2 19840.158} C_VEL
LIN {X 0,Y 439.161,Z 712.844,A -85,B 0,C 180,E1 19838.658,E2 19838.658} C_VEL
LIN {X 0,Y 441.357,Z 695.405,A -85,B 0,C 180,E1 19837.333,E2 19837.333} C_VEL
LIN {X 0,Y 443.348,Z 677.002,A -85,B 0,C 180,E1 19836.218,E2 19836.218} C_VEL
LIN {X 0,Y 445.086,Z 657.689,A -85,B 0,C 180,E1 19835.322,E2 19835.322} C_VEL
LIN {X 0,Y 446.461,Z 637.978,A -85,B 0,C 180,E1 19834.664,E2 19834.664} C_VEL
LIN {X 0,Y 447.657,Z 611.22,A -85,B 0,C 180,E1 19834.091,E2 19834.091} C_VEL
LIN {X 0,Y 453.944,Z 441.845,A -85,B 0,C 180,E1 19830.892,E2 19830.892} C_VEL
LIN {X 0,Y 449.362,Z 398.087,A -85,B 0,C 180,E1 19829.286,E2 19829.286} C_VEL
LIN {X 0,Y 455.487,Z 340.396,A -85,B 0,C 180,E1 19825.065,E2 19825.065} C_VEL
LIN {X 0,Y 458.821,Z 310.4,A -85,B 0,C 180,E1 19822.815,E2 19822.815} C_VEL
LIN {X 0,Y 451.781,Z 294.89,A -85,B 0,C 180,E1 19820.332,E2 19820.332} C_VEL
LIN {X 0,Y 444.419,Z 279.976,A -85,B 0,C 180,E1 19817.613,E2 19817.613} C_VEL
LIN {X 0,Y 439.122,Z 270.362,A -85,B 0,C 180,E1 19815.585,E2 19815.585} C_VEL
LIN {X 0,Y 436.338,Z 265.444,A -85,B 0,C 180,E1 19814.463,E2 19814.463} C_VEL
LIN {X 0,Y 434.316,Z 261.67,A -85,B 0,C 180,E1 19813.58,E2 19813.58} C_VEL
LIN {X 0,Y 431.97,Z 257.671,A -85,B 0,C 180,E1 19812.566,E2 19812.566} C_VEL
LIN {X 0,Y 430.716,Z 255.937,A -85,B 0,C 180,E1 19812.059,E2 19812.059} C_VEL
LIN {X 0,Y 428.836,Z 252.553,A -85,B 0,C 180,E1 19811.158,E2 19811.158} C_VEL
LIN {X 0,Y 428.043,Z 251.17,A -85,B 0,C 180,E1 19810.77,E2 19810.77} C_VEL
